KUKA KRL program: f1_Kuka_APT222T03S22.SRC

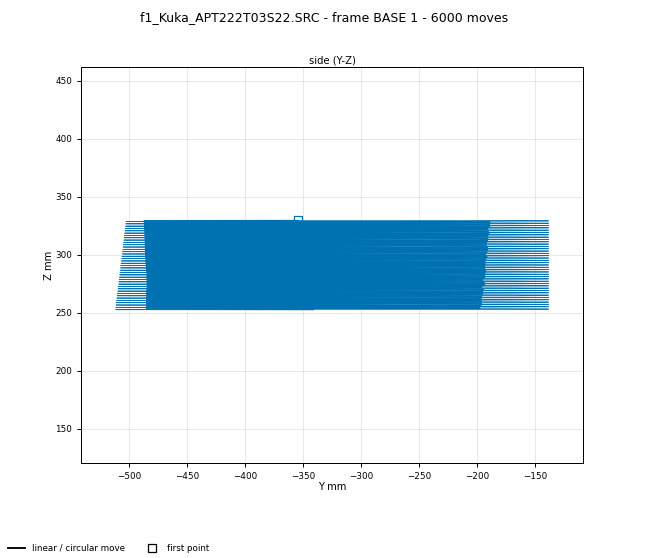
[picture p0: tool path of f1_Kuka_APT222T03S22.SRC in frame BASE 1, 6000 of 6001 moves have a stored position in this frame; points joined in program order, loops and branches not executed]
&ACCESS RVP
&REL 2
&PARAM TEMPLATE = C:\KRC\Roboter\Template\vorgabe
&PARAM EDITMASK = *
DEF f1_Kuka_APT222T03S22()


;FOLD INI;%{PE}%V3.2.0,%MKUKATPBASIS,%CINIT,%VCOMMON,%P
  ;FOLD BAS INI;%{E}%V3.2.0,%MKUKATPBASIS,%CINIT,%VINIT,%P
    GLOBAL INTERRUPT DECL 3 WHEN $STOPMESS==TRUE DO IR_STOPM ( )
    INTERRUPT ON 3
    BAS (#INITMOV,0 )
  ;ENDFOLD (BAS INI)
  ;FOLD USER INI;%{E}%V3.2.0,%MKUKATPUSER,%CINIT,%VINIT,%P
    ;Make your modifications here
  ;ENDFOLD (USER INI)
;ENDFOLD (INI)


;*** Make Null PTP Move
  PTP $pos_act

;*** Auto Load The Correct TOOL Data
  $tool=tool_data[3]

;*** Auto Load The Correct BASE Data
  $base=base_data[1]

  $ADVANCE = 5

;*** Restate Last Velocity
MMPM(30000.0)
SetRPM(6000)
LIN {X -0.045,Y -354.081,Z 329.624,A 0.000,B 0.000,C 90.000,E1 292.333} C_DIS
LIN {X -0.124,Y -370.125,Z 329.612,A 0.000,B 0.000,C 90.000,E1 290.248} C_DIS
LIN {X -0.194,Y -391.997,Z 329.598,A 0.000,B 0.000,C 90.000,E1 287.638} C_DIS
LIN {X 0.138,Y -406.942,Z 329.588,A 0.000,B 0.000,C 90.000,E1 285.898} C_DIS
LIN {X -0.099,Y -421.524,Z 329.579,A 0.000,B 0.000,C 90.000,E1 284.300} C_DIS
LIN {X 0.209,Y -431.131,Z 329.573,A 0.000,B 0.000,C 90.000,E1 283.175} C_DIS
LIN {X -0.088,Y -437.715,Z 329.569,A 0.000,B 0.000,C 90.000,E1 282.411} C_DIS
LIN {X -0.210,Y -445.768,Z 329.563,A 0.000,B 0.000,C 90.000,E1 281.366} C_DIS
LIN {X -0.147,Y -453.240,Z 329.557,A 0.000,B 0.000,C 90.000,E1 280.310} C_DIS
LIN {X -0.080,Y -460.078,Z 329.551,A 0.000,B 0.000,C 90.000,E1 279.265} C_DIS
LIN {X -0.164,Y -468.020,Z 329.544,A 0.000,B 0.000,C 90.000,E1 277.992} C_DIS
LIN {X 0.077,Y -473.919,Z 329.539,A 0.000,B 0.000,C 90.000,E1 276.947} C_DIS
LIN {X -0.147,Y -479.234,Z 329.533,A 0.000,B 0.000,C 90.000,E1 275.967} C_DIS
LIN {X -0.044,Y -481.494,Z 329.530,A 0.000,B 0.000,C 90.000,E1 275.454} C_DIS
LIN {X 0.122,Y -483.441,Z 329.527,A 0.000,B 0.000,C 90.000,E1 274.935} C_DIS
LIN {X -0.189,Y -484.967,Z 329.525,A 0.000,B 0.000,C 90.000,E1 274.473} C_DIS
LIN {X -0.009,Y -486.097,Z 329.522,A 0.000,B 0.000,C 90.000,E1 273.955} C_DIS
LIN {X 0.148,Y -486.777,Z 329.519,A 0.000,B 0.000,C 90.000,E1 273.440} C_DIS
LIN {X -0.146,Y -487.135,Z 329.516,A 0.000,B 0.000,C 90.000,E1 272.980} C_DIS
LIN {X 0.025,Y -487.164,Z 329.514,A 0.000,B 0.000,C 90.000,E1 272.465} C_DIS
LIN {X -0.093,Y -486.656,Z 329.508,A 0.000,B 0.000,C 90.000,E1 271.489} C_DIS
LIN {X 0.082,Y -486.195,Z 329.505,A 0.000,B 0.000,C 90.000,E1 270.974} C_DIS
LIN {X -0.228,Y -485.501,Z 329.503,A 0.000,B 0.000,C 90.000,E1 270.516} C_DIS
LIN {X -0.056,Y -484.497,Z 329.500,A 0.000,B 0.000,C 90.000,E1 270.000} C_DIS
LIN {X 0.112,Y -482.951,Z 329.497,A 0.000,B 0.000,C 90.000,E1 269.484} C_DIS
LIN {X -0.209,Y -480.802,Z 329.494,A 0.000,B 0.000,C 90.000,E1 269.026} C_DIS
LIN {X -0.057,Y -477.885,Z 329.492,A 0.000,B 0.000,C 90.000,E1 268.511} C_DIS
LIN {X -0.231,Y -476.129,Z 329.490,A 0.000,B 0.000,C 90.000,E1 268.282} C_DIS
LIN {X 0.087,Y -474.110,Z 329.489,A 0.000,B 0.000,C 90.000,E1 267.993} C_DIS
LIN {X 0.195,Y -469.213,Z 329.486,A 0.000,B 0.000,C 90.000,E1 267.478} C_DIS
LIN {X 0.065,Y -466.330,Z 329.485,A 0.000,B 0.000,C 90.000,E1 267.249} C_DIS
LIN {X -0.065,Y -463.081,Z 329.483,A 0.000,B 0.000,C 90.000,E1 267.020} C_DIS
LIN {X 0.146,Y -459.910,Z 329.482,A 0.000,B 0.000,C 90.000,E1 266.788} C_DIS
LIN {X -0.126,Y -456.229,Z 329.481,A 0.000,B 0.000,C 90.000,E1 266.617} C_DIS
LIN {X -0.058,Y -452.834,Z 329.480,A 0.000,B 0.000,C 90.000,E1 266.445} C_DIS
LIN {X -0.061,Y -445.345,Z 329.479,A 0.000,B 0.000,C 90.000,E1 266.159} C_DIS
LIN {X 0.071,Y -437.546,Z 329.477,A 0.000,B 0.000,C 90.000,E1 265.927} C_DIS
LIN {X 0.203,Y -429.002,Z 329.477,A 0.000,B 0.000,C 90.000,E1 265.755} C_DIS
LIN {X 0.032,Y -418.844,Z 329.476,A 0.000,B 0.000,C 90.000,E1 265.698} C_DIS
LIN {X -0.015,Y -180.910,Z 329.476,A 0.000,B 0.000,C 90.000,E1 265.698} C_DIS
LIN {X 0.075,Y -180.806,Z 329.471,A 0.000,B 0.000,C 90.000,E1 264.780} C_DIS
LIN {X -0.027,Y -178.907,Z 329.443,A 0.000,B 0.000,C 90.000,E1 259.746} C_DIS
LIN {X 0.053,Y -175.951,Z 329.415,A 0.000,B 0.000,C 90.000,E1 254.629} C_DIS
LIN {X 0.000,Y -175.416,Z 329.410,A 0.000,B 0.000,C 90.000,E1 253.795} C_DIS
LIN {X 0.003,Y -172.179,Z 329.386,A 0.000,B 0.000,C 90.000,E1 249.518} C_DIS
LIN {X 0.042,Y -171.650,Z 329.381,A 0.000,B 0.000,C 90.000,E1 248.646} C_DIS
LIN {X 0.036,Y -167.874,Z 329.357,A 0.000,B 0.000,C 90.000,E1 244.332} C_DIS
LIN {X -0.021,Y -166.608,Z 329.348,A 0.000,B 0.000,C 90.000,E1 242.615} C_DIS
LIN {X -0.027,Y -162.597,Z 329.324,A 0.000,B 0.000,C 90.000,E1 238.250} C_DIS
LIN {X -0.053,Y -161.281,Z 329.314,A 0.000,B 0.000,C 90.000,E1 236.501} C_DIS
LIN {X -0.017,Y -157.280,Z 329.289,A 0.000,B 0.000,C 90.000,E1 232.065} C_DIS
LIN {X 0.006,Y -155.999,Z 329.279,A 0.000,B 0.000,C 90.000,E1 230.275} C_DIS
LIN {X -0.034,Y -152.257,Z 329.254,A 0.000,B 0.000,C 90.000,E1 225.810} C_DIS
LIN {X -0.012,Y -150.495,Z 329.239,A 0.000,B 0.000,C 90.000,E1 223.095} C_DIS
LIN {X 0.018,Y -147.219,Z 329.214,A 0.000,B 0.000,C 90.000,E1 218.543} C_DIS
LIN {X -0.013,Y -145.241,Z 329.194,A 0.000,B 0.000,C 90.000,E1 214.898} C_DIS
LIN {X 0.029,Y -142.362,Z 329.163,A 0.000,B 0.000,C 90.000,E1 209.361} C_DIS
LIN {X 0.025,Y -141.748,Z 329.153,A 0.000,B 0.000,C 90.000,E1 207.513} C_DIS
LIN {X -0.048,Y -139.492,Z 329.117,A 0.000,B 0.000,C 90.000,E1 201.046} C_DIS
LIN {X -0.012,Y -138.995,Z 329.101,A 0.000,B 0.000,C 90.000,E1 198.236} C_DIS
LIN {X -0.055,Y -138.336,Z 329.055,A 0.000,B 0.000,C 90.000,E1 189.849} C_DIS
LIN {X -0.033,Y -139.415,Z 329.008,A 0.000,B 0.000,C 90.000,E1 181.432} C_DIS
LIN {X 0.021,Y -141.329,Z 328.972,A 0.000,B 0.000,C 90.000,E1 174.894} C_DIS
LIN {X -0.022,Y -142.686,Z 328.956,A 0.000,B 0.000,C 90.000,E1 172.129} C_DIS
LIN {X -0.043,Y -145.046,Z 328.931,A 0.000,B 0.000,C 90.000,E1 167.521} C_DIS
LIN {X -0.046,Y -147.673,Z 328.910,A 0.000,B 0.000,C 90.000,E1 163.850} C_DIS
LIN {X -0.011,Y -150.315,Z 328.890,A 0.000,B 0.000,C 90.000,E1 160.188} C_DIS
LIN {X 0.061,Y -153.728,Z 328.870,A 0.000,B 0.000,C 90.000,E1 156.538} C_DIS
LIN {X -0.087,Y -157.141,Z 328.850,A 0.000,B 0.000,C 90.000,E1 152.999} C_DIS
LIN {X -0.013,Y -161.290,Z 328.830,A 0.000,B 0.000,C 90.000,E1 149.410} C_DIS
LIN {X 0.004,Y -164.406,Z 328.815,A 0.000,B 0.000,C 90.000,E1 146.755} C_DIS
LIN {X 0.001,Y -169.087,Z 328.796,A 0.000,B 0.000,C 90.000,E1 143.256} C_DIS
LIN {X -0.048,Y -171.643,Z 328.786,A 0.000,B 0.000,C 90.000,E1 141.537} C_DIS
LIN {X -0.001,Y -176.606,Z 328.767,A 0.000,B 0.000,C 90.000,E1 138.081} C_DIS
LIN {X 0.000,Y -180.905,Z 328.753,A 0.000,B 0.000,C 90.000,E1 135.526} C_DIS
LIN {X -0.009,Y -186.320,Z 328.734,A 0.000,B 0.000,C 90.000,E1 132.162} C_DIS
LIN {X 0.058,Y -190.954,Z 328.720,A 0.000,B 0.000,C 90.000,E1 129.644} C_DIS
LIN {X -0.022,Y -196.725,Z 328.702,A 0.000,B 0.000,C 90.000,E1 126.377} C_DIS
LIN {X -0.054,Y -201.183,Z 328.689,A 0.000,B 0.000,C 90.000,E1 124.119} C_DIS
LIN {X -0.051,Y -201.261,Z 328.689,A 0.000,B 0.000,C 90.000,E1 124.072} C_DIS
LIN {X 0.058,Y -302.172,Z 328.689,A 0.000,B 0.000,C 90.000,E1 124.040} C_DIS
LIN {X 0.097,Y -306.283,Z 328.689,A 0.000,B 0.000,C 90.000,E1 123.913} C_DIS
LIN {X -0.045,Y -309.181,Z 328.687,A 0.000,B 0.000,C 90.000,E1 123.754} C_DIS
LIN {X -0.078,Y -312.923,Z 328.685,A 0.000,B 0.000,C 90.000,E1 123.372} C_DIS
LIN {X 0.156,Y -316.425,Z 328.682,A 0.000,B 0.000,C 90.000,E1 122.752} C_DIS
LIN {X 0.006,Y -318.957,Z 328.679,A 0.000,B 0.000,C 90.000,E1 122.133} C_DIS
LIN {X -0.076,Y -329.793,Z 328.663,A 0.000,B 0.000,C 90.000,E1 119.283} C_DIS
LIN {X -0.172,Y -342.027,Z 328.647,A 0.000,B 0.000,C 90.000,E1 116.488} C_DIS
LIN {X -0.094,Y -354.161,Z 328.633,A 0.000,B 0.000,C 90.000,E1 114.027} C_DIS
LIN {X 0.155,Y -367.575,Z 328.620,A 0.000,B 0.000,C 90.000,E1 111.589} C_DIS
LIN {X -0.007,Y -382.364,Z 328.607,A 0.000,B 0.000,C 90.000,E1 109.268} C_DIS
LIN {X -0.052,Y -398.640,Z 328.594,A 0.000,B 0.000,C 90.000,E1 106.985} C_DIS
LIN {X -0.199,Y -416.523,Z 328.582,A 0.000,B 0.000,C 90.000,E1 104.773} C_DIS
LIN {X -0.055,Y -436.052,Z 328.570,A 0.000,B 0.000,C 90.000,E1 102.591} C_DIS
LIN {X -0.147,Y -456.379,Z 328.559,A 0.000,B 0.000,C 90.000,E1 100.602} C_DIS
LIN {X 0.183,Y -479.856,Z 328.547,A 0.000,B 0.000,C 90.000,E1 98.511} C_DIS
LIN {X -0.219,Y -495.644,Z 328.540,A 0.000,B 0.000,C 90.000,E1 97.296} C_DIS
LIN {X -0.016,Y -497.526,Z 328.539,A 0.000,B 0.000,C 90.000,E1 97.068} C_DIS
LIN {X -0.103,Y -499.247,Z 328.538,A 0.000,B 0.000,C 90.000,E1 96.834} C_DIS
LIN {X -0.251,Y -500.536,Z 328.537,A 0.000,B 0.000,C 90.000,E1 96.606} C_DIS
LIN {X 0.032,Y -502.123,Z 328.534,A 0.000,B 0.000,C 90.000,E1 96.087} C_DIS
LIN {X -0.178,Y -502.633,Z 328.531,A 0.000,B 0.000,C 90.000,E1 95.625} C_DIS
LIN {X 0.120,Y -502.144,Z 328.528,A 0.000,B 0.000,C 90.000,E1 95.106} C_DIS
LIN {X -0.081,Y -500.573,Z 328.526,A 0.000,B 0.000,C 90.000,E1 94.645} C_DIS
LIN {X -0.202,Y -499.293,Z 328.524,A 0.000,B 0.000,C 90.000,E1 94.416} C_DIS
LIN {X -0.045,Y -494.012,Z 328.520,A 0.000,B 0.000,C 90.000,E1 93.669} C_DIS
LIN {X -0.084,Y -486.242,Z 328.515,A 0.000,B 0.000,C 90.000,E1 92.694} C_DIS
LIN {X -0.157,Y -467.875,Z 328.502,A 0.000,B 0.000,C 90.000,E1 90.458} C_DIS
LIN {X 0.002,Y -448.883,Z 328.488,A 0.000,B 0.000,C 90.000,E1 87.879} C_DIS
LIN {X -0.168,Y -430.026,Z 328.472,A 0.000,B 0.000,C 90.000,E1 85.008} C_DIS
LIN {X -0.089,Y -414.527,Z 328.457,A 0.000,B 0.000,C 90.000,E1 82.299} C_DIS
LIN {X 0.114,Y -399.996,Z 328.442,A 0.000,B 0.000,C 90.000,E1 79.511} C_DIS
LIN {X -0.212,Y -389.916,Z 328.431,A 0.000,B 0.000,C 90.000,E1 77.589} C_DIS
LIN {X -0.081,Y -378.252,Z 328.418,A 0.000,B 0.000,C 90.000,E1 75.283} C_DIS
LIN {X -0.109,Y -368.106,Z 328.407,A 0.000,B 0.000,C 90.000,E1 73.251} C_DIS
LIN {X 0.100,Y -357.919,Z 328.395,A 0.000,B 0.000,C 90.000,E1 71.148} C_DIS
LIN {X -0.103,Y -346.247,Z 328.382,A 0.000,B 0.000,C 90.000,E1 68.773} C_DIS
LIN {X 0.108,Y -333.824,Z 328.367,A 0.000,B 0.000,C 90.000,E1 65.973} C_DIS
LIN {X -0.011,Y -320.451,Z 328.347,A 0.000,B 0.000,C 90.000,E1 62.538} C_DIS
LIN {X -0.030,Y -309.036,Z 328.330,A 0.000,B 0.000,C 90.000,E1 59.331} C_DIS
LIN {X 0.011,Y -297.294,Z 328.310,A 0.000,B 0.000,C 90.000,E1 55.722} C_DIS
LIN {X -0.049,Y -287.389,Z 328.291,A 0.000,B 0.000,C 90.000,E1 52.396} C_DIS
LIN {X 0.036,Y -279.768,Z 328.276,A 0.000,B 0.000,C 90.000,E1 49.666} C_DIS
LIN {X -0.101,Y -274.008,Z 328.265,A 0.000,B 0.000,C 90.000,E1 47.634} C_DIS
LIN {X -0.035,Y -266.352,Z 328.249,A 0.000,B 0.000,C 90.000,E1 44.838} C_DIS
LIN {X 0.122,Y -260.736,Z 328.237,A 0.000,B 0.000,C 90.000,E1 42.690} C_DIS
LIN {X -0.176,Y -255.046,Z 328.225,A 0.000,B 0.000,C 90.000,E1 40.620} C_DIS
LIN {X 0.006,Y -249.323,Z 328.213,A 0.000,B 0.000,C 90.000,E1 38.418} C_DIS
LIN {X 0.075,Y -243.454,Z 328.201,A 0.000,B 0.000,C 90.000,E1 36.217} C_DIS
LIN {X -0.050,Y -235.570,Z 328.185,A 0.000,B 0.000,C 90.000,E1 33.293} C_DIS
LIN {X 0.092,Y -227.992,Z 328.168,A 0.000,B 0.000,C 90.000,E1 30.256} C_DIS
LIN {X -0.098,Y -220.827,Z 328.151,A 0.000,B 0.000,C 90.000,E1 27.257} C_DIS
LIN {X 0.024,Y -214.294,Z 328.134,A 0.000,B 0.000,C 90.000,E1 24.131} C_DIS
LIN {X 0.107,Y -208.616,Z 328.117,A 0.000,B 0.000,C 90.000,E1 20.972} C_DIS
LIN {X -0.040,Y -202.573,Z 328.095,A 0.000,B 0.000,C 90.000,E1 17.040} C_DIS
LIN {X -0.053,Y -198.494,Z 328.077,A 0.000,B 0.000,C 90.000,E1 13.828} C_DIS
LIN {X 0.096,Y -194.493,Z 328.054,A 0.000,B 0.000,C 90.000,E1 9.726} C_DIS
LIN {X 0.063,Y -191.104,Z 328.027,A 0.000,B 0.000,C 90.000,E1 4.821} C_DIS
LIN {X -0.006,Y -188.880,Z 327.988,A 0.000,B 0.000,C 90.000,E1 357.879} C_DIS
LIN {X 0.038,Y -190.678,Z 327.933,A 0.000,B 0.000,C 90.000,E1 347.937} C_DIS
LIN {X -0.017,Y -193.867,Z 327.906,A 0.000,B 0.000,C 90.000,E1 343.015} C_DIS
LIN {X 0.080,Y -197.691,Z 327.883,A 0.000,B 0.000,C 90.000,E1 338.901} C_DIS
LIN {X 0.105,Y -202.533,Z 327.860,A 0.000,B 0.000,C 90.000,E1 334.845} C_DIS
LIN {X -0.015,Y -208.379,Z 327.838,A 0.000,B 0.000,C 90.000,E1 330.873} C_DIS
LIN {X 0.008,Y -215.221,Z 327.816,A 0.000,B 0.000,C 90.000,E1 326.914} C_DIS
LIN {X 0.068,Y -222.764,Z 327.795,A 0.000,B 0.000,C 90.000,E1 323.004} C_DIS
LIN {X -0.004,Y -229.499,Z 327.777,A 0.000,B 0.000,C 90.000,E1 319.952} C_DIS
LIN {X 0.045,Y -238.222,Z 327.759,A 0.000,B 0.000,C 90.000,E1 316.539} C_DIS
LIN {X 0.014,Y -247.221,Z 327.742,A 0.000,B 0.000,C 90.000,E1 313.581} C_DIS
LIN {X 0.069,Y -258.416,Z 327.724,A 0.000,B 0.000,C 90.000,E1 310.297} C_DIS
LIN {X 0.015,Y -270.485,Z 327.706,A 0.000,B 0.000,C 90.000,E1 307.111} C_DIS
LIN {X -0.011,Y -279.232,Z 327.695,A 0.000,B 0.000,C 90.000,E1 305.025} C_DIS
LIN {X 0.126,Y -293.754,Z 327.678,A 0.000,B 0.000,C 90.000,E1 301.926} C_DIS
LIN {X 0.079,Y -309.866,Z 327.661,A 0.000,B 0.000,C 90.000,E1 298.949} C_DIS
LIN {X 0.106,Y -321.655,Z 327.650,A 0.000,B 0.000,C 90.000,E1 297.001} C_DIS
LIN {X -0.144,Y -338.816,Z 327.636,A 0.000,B 0.000,C 90.000,E1 294.515} C_DIS
LIN {X 0.065,Y -356.624,Z 327.622,A 0.000,B 0.000,C 90.000,E1 292.025} C_DIS
LIN {X 0.136,Y -375.134,Z 327.609,A 0.000,B 0.000,C 90.000,E1 289.631} C_DIS
LIN {X -0.123,Y -396.978,Z 327.595,A 0.000,B 0.000,C 90.000,E1 287.094} C_DIS
LIN {X -0.204,Y -411.779,Z 327.586,A 0.000,B 0.000,C 90.000,E1 285.426} C_DIS
LIN {X -0.152,Y -426.487,Z 327.576,A 0.000,B 0.000,C 90.000,E1 283.772} C_DIS
LIN {X 0.085,Y -433.401,Z 327.572,A 0.000,B 0.000,C 90.000,E1 282.939} C_DIS
LIN {X 0.004,Y -441.777,Z 327.566,A 0.000,B 0.000,C 90.000,E1 281.883} C_DIS
LIN {X -0.067,Y -449.482,Z 327.560,A 0.000,B 0.000,C 90.000,E1 280.838} C_DIS
LIN {X -0.040,Y -456.608,Z 327.554,A 0.000,B 0.000,C 90.000,E1 279.792} C_DIS
LIN {X -0.101,Y -464.753,Z 327.547,A 0.000,B 0.000,C 90.000,E1 278.511} C_DIS
LIN {X 0.041,Y -470.830,Z 327.542,A 0.000,B 0.000,C 90.000,E1 277.473} C_DIS
LIN {X -0.156,Y -476.468,Z 327.536,A 0.000,B 0.000,C 90.000,E1 276.486} C_DIS
LIN {X -0.213,Y -480.238,Z 327.532,A 0.000,B 0.000,C 90.000,E1 275.739} C_DIS
LIN {X -0.237,Y -483.273,Z 327.528,A 0.000,B 0.000,C 90.000,E1 274.992} C_DIS
LIN {X -0.068,Y -484.803,Z 327.525,A 0.000,B 0.000,C 90.000,E1 274.473} C_DIS
LIN {X 0.111,Y -485.920,Z 327.522,A 0.000,B 0.000,C 90.000,E1 273.955} C_DIS
LIN {X -0.219,Y -486.610,Z 327.519,A 0.000,B 0.000,C 90.000,E1 273.498} C_DIS
LIN {X -0.028,Y -486.989,Z 327.517,A 0.000,B 0.000,C 90.000,E1 272.980} C_DIS
LIN {X 0.142,Y -487.029,Z 327.514,A 0.000,B 0.000,C 90.000,E1 272.465} C_DIS
LIN {X 0.023,Y -486.519,Z 327.508,A 0.000,B 0.000,C 90.000,E1 271.489} C_DIS
LIN {X 0.197,Y -486.074,Z 327.506,A 0.000,B 0.000,C 90.000,E1 270.974} C_DIS
LIN {X -0.114,Y -485.390,Z 327.503,A 0.000,B 0.000,C 90.000,E1 270.516} C_DIS
LIN {X 0.057,Y -484.402,Z 327.500,A 0.000,B 0.000,C 90.000,E1 270.000} C_DIS
LIN {X 0.224,Y -482.871,Z 327.497,A 0.000,B 0.000,C 90.000,E1 269.484} C_DIS
LIN {X -0.097,Y -480.780,Z 327.495,A 0.000,B 0.000,C 90.000,E1 269.026} C_DIS
LIN {X 0.053,Y -477.912,Z 327.492,A 0.000,B 0.000,C 90.000,E1 268.511} C_DIS
LIN {X 0.196,Y -474.183,Z 327.489,A 0.000,B 0.000,C 90.000,E1 267.993} C_DIS
LIN {X -0.166,Y -469.376,Z 327.486,A 0.000,B 0.000,C 90.000,E1 267.535} C_DIS
LIN {X 0.163,Y -466.544,Z 327.485,A 0.000,B 0.000,C 90.000,E1 267.249} C_DIS
LIN {X 0.025,Y -463.317,Z 327.483,A 0.000,B 0.000,C 90.000,E1 267.020} C_DIS
LIN {X 0.223,Y -460.234,Z 327.482,A 0.000,B 0.000,C 90.000,E1 266.788} C_DIS
LIN {X -0.064,Y -456.610,Z 327.481,A 0.000,B 0.000,C 90.000,E1 266.617} C_DIS
LIN {X -0.022,Y -453.219,Z 327.480,A 0.000,B 0.000,C 90.000,E1 266.445} C_DIS
LIN {X -0.073,Y -445.673,Z 327.479,A 0.000,B 0.000,C 90.000,E1 266.159} C_DIS
LIN {X 0.032,Y -437.850,Z 327.477,A 0.000,B 0.000,C 90.000,E1 265.927} C_DIS
LIN {X 0.145,Y -429.297,Z 327.477,A 0.000,B 0.000,C 90.000,E1 265.755} C_DIS
LIN {X -0.046,Y -419.572,Z 327.476,A 0.000,B 0.000,C 90.000,E1 265.698} C_DIS
LIN {X -0.114,Y -416.030,Z 327.476,A 0.000,B 0.000,C 90.000,E1 265.698} C_DIS
LIN {X -0.081,Y -180.910,Z 327.476,A 0.000,B 0.000,C 90.000,E1 265.698} C_DIS
LIN {X 0.037,Y -180.802,Z 327.471,A 0.000,B 0.000,C 90.000,E1 264.780} C_DIS
LIN {X -0.066,Y -178.902,Z 327.443,A 0.000,B 0.000,C 90.000,E1 259.746} C_DIS
LIN {X 0.015,Y -175.945,Z 327.415,A 0.000,B 0.000,C 90.000,E1 254.629} C_DIS
LIN {X -0.039,Y -175.405,Z 327.410,A 0.000,B 0.000,C 90.000,E1 253.795} C_DIS
LIN {X -0.036,Y -172.171,Z 327.386,A 0.000,B 0.000,C 90.000,E1 249.518} C_DIS
LIN {X 0.004,Y -171.641,Z 327.381,A 0.000,B 0.000,C 90.000,E1 248.646} C_DIS
LIN {X -0.001,Y -167.864,Z 327.357,A 0.000,B 0.000,C 90.000,E1 244.332} C_DIS
LIN {X -0.058,Y -166.597,Z 327.348,A 0.000,B 0.000,C 90.000,E1 242.615} C_DIS
LIN {X 0.075,Y -162.587,Z 327.323,A 0.000,B 0.000,C 90.000,E1 238.201} C_DIS
LIN {X -0.089,Y -161.271,Z 327.314,A 0.000,B 0.000,C 90.000,E1 236.501} C_DIS
LIN {X 0.043,Y -157.270,Z 327.289,A 0.000,B 0.000,C 90.000,E1 232.029} C_DIS
LIN {X -0.030,Y -155.990,Z 327.279,A 0.000,B 0.000,C 90.000,E1 230.275} C_DIS
LIN {X -0.069,Y -152.247,Z 327.254,A 0.000,B 0.000,C 90.000,E1 225.810} C_DIS
LIN {X -0.047,Y -150.487,Z 327.239,A 0.000,B 0.000,C 90.000,E1 223.095} C_DIS
LIN {X -0.016,Y -147.211,Z 327.214,A 0.000,B 0.000,C 90.000,E1 218.543} C_DIS
LIN {X -0.047,Y -145.232,Z 327.194,A 0.000,B 0.000,C 90.000,E1 214.898} C_DIS
LIN {X 0.065,Y -142.356,Z 327.163,A 0.000,B 0.000,C 90.000,E1 209.333} C_DIS
LIN {X -0.008,Y -141.743,Z 327.153,A 0.000,B 0.000,C 90.000,E1 207.513} C_DIS
LIN {X -0.032,Y -139.489,Z 327.117,A 0.000,B 0.000,C 90.000,E1 201.025} C_DIS
LIN {X -0.044,Y -138.992,Z 327.101,A 0.000,B 0.000,C 90.000,E1 198.236} C_DIS
LIN {X 0.048,Y -138.336,Z 327.055,A 0.000,B 0.000,C 90.000,E1 189.792} C_DIS
LIN {X -0.066,Y -139.418,Z 327.008,A 0.000,B 0.000,C 90.000,E1 181.432} C_DIS
LIN {X -0.013,Y -141.335,Z 326.972,A 0.000,B 0.000,C 90.000,E1 174.894} C_DIS
LIN {X -0.056,Y -142.691,Z 326.956,A 0.000,B 0.000,C 90.000,E1 172.129} C_DIS
LIN {X 0.065,Y -145.055,Z 326.931,A 0.000,B 0.000,C 90.000,E1 167.465} C_DIS
LIN {X 0.062,Y -147.680,Z 326.910,A 0.000,B 0.000,C 90.000,E1 163.795} C_DIS
LIN {X -0.046,Y -150.326,Z 326.890,A 0.000,B 0.000,C 90.000,E1 160.188} C_DIS
LIN {X 0.025,Y -153.742,Z 326.870,A 0.000,B 0.000,C 90.000,E1 156.538} C_DIS
LIN {X 0.017,Y -157.155,Z 326.850,A 0.000,B 0.000,C 90.000,E1 152.948} C_DIS
LIN {X -0.049,Y -161.307,Z 326.830,A 0.000,B 0.000,C 90.000,E1 149.410} C_DIS
LIN {X -0.032,Y -164.422,Z 326.815,A 0.000,B 0.000,C 90.000,E1 146.755} C_DIS
LIN {X -0.036,Y -169.106,Z 326.796,A 0.000,B 0.000,C 90.000,E1 143.256} C_DIS
LIN {X -0.085,Y -171.661,Z 326.786,A 0.000,B 0.000,C 90.000,E1 141.537} C_DIS
LIN {X -0.040,Y -176.626,Z 326.767,A 0.000,B 0.000,C 90.000,E1 138.081} C_DIS
LIN {X 0.088,Y -180.923,Z 326.753,A 0.000,B 0.000,C 90.000,E1 135.486} C_DIS
LIN {X -0.049,Y -186.342,Z 326.734,A 0.000,B 0.000,C 90.000,E1 132.162} C_DIS
LIN {X 0.018,Y -190.974,Z 326.720,A 0.000,B 0.000,C 90.000,E1 129.644} C_DIS
LIN {X -0.063,Y -196.749,Z 326.702,A 0.000,B 0.000,C 90.000,E1 126.377} C_DIS
LIN {X -0.012,Y -201.162,Z 326.690,A 0.000,B 0.000,C 90.000,E1 124.119} C_DIS
LIN {X 0.012,Y -201.366,Z 326.689,A 0.000,B 0.000,C 90.000,E1 123.992} C_DIS
LIN {X -0.018,Y -302.297,Z 326.689,A 0.000,B 0.000,C 90.000,E1 123.992} C_DIS
LIN {X 0.034,Y -305.307,Z 326.688,A 0.000,B 0.000,C 90.000,E1 123.913} C_DIS
LIN {X -0.183,Y -308.457,Z 326.688,A 0.000,B 0.000,C 90.000,E1 123.785} C_DIS
LIN {X 0.025,Y -312.067,Z 326.686,A 0.000,B 0.000,C 90.000,E1 123.420} C_DIS
LIN {X 0.137,Y -315.668,Z 326.683,A 0.000,B 0.000,C 90.000,E1 122.880} C_DIS
LIN {X 0.193,Y -317.253,Z 326.681,A 0.000,B 0.000,C 90.000,E1 122.546} C_DIS
LIN {X -0.013,Y -330.566,Z 326.662,A 0.000,B 0.000,C 90.000,E1 119.077} C_DIS
LIN {X -0.087,Y -342.897,Z 326.646,A 0.000,B 0.000,C 90.000,E1 116.283} C_DIS
LIN {X 0.009,Y -355.126,Z 326.632,A 0.000,B 0.000,C 90.000,E1 113.823} C_DIS
LIN {X 0.143,Y -368.642,Z 326.619,A 0.000,B 0.000,C 90.000,E1 111.408} C_DIS
LIN {X 0.008,Y -383.542,Z 326.606,A 0.000,B 0.000,C 90.000,E1 109.087} C_DIS
LIN {X -0.005,Y -399.937,Z 326.593,A 0.000,B 0.000,C 90.000,E1 106.804} C_DIS
LIN {X -0.121,Y -417.949,Z 326.581,A 0.000,B 0.000,C 90.000,E1 104.592} C_DIS
LIN {X 0.097,Y -437.567,Z 326.569,A 0.000,B 0.000,C 90.000,E1 102.411} C_DIS
LIN {X 0.028,Y -457.937,Z 326.558,A 0.000,B 0.000,C 90.000,E1 100.433} C_DIS
LIN {X -0.006,Y -481.486,Z 326.547,A 0.000,B 0.000,C 90.000,E1 98.398} C_DIS
LIN {X -0.044,Y -494.774,Z 326.541,A 0.000,B 0.000,C 90.000,E1 97.352} C_DIS
LIN {X 0.152,Y -496.923,Z 326.540,A 0.000,B 0.000,C 90.000,E1 97.125} C_DIS
LIN {X 0.147,Y -498.786,Z 326.538,A 0.000,B 0.000,C 90.000,E1 96.891} C_DIS
LIN {X 0.081,Y -500.200,Z 326.537,A 0.000,B 0.000,C 90.000,E1 96.663} C_DIS
LIN {X -0.137,Y -502.077,Z 326.534,A 0.000,B 0.000,C 90.000,E1 96.201} C_DIS
LIN {X 0.151,Y -502.826,Z 326.532,A 0.000,B 0.000,C 90.000,E1 95.682} C_DIS
LIN {X -0.052,Y -502.569,Z 326.529,A 0.000,B 0.000,C 90.000,E1 95.220} C_DIS
LIN {X 0.246,Y -501.265,Z 326.526,A 0.000,B 0.000,C 90.000,E1 94.702} C_DIS
LIN {X 0.125,Y -500.154,Z 326.525,A 0.000,B 0.000,C 90.000,E1 94.473} C_DIS
LIN {X 0.005,Y -498.656,Z 326.524,A 0.000,B 0.000,C 90.000,E1 94.245} C_DIS
LIN {X 0.020,Y -491.314,Z 326.518,A 0.000,B 0.000,C 90.000,E1 93.269} C_DIS
LIN {X -0.047,Y -483.293,Z 326.513,A 0.000,B 0.000,C 90.000,E1 92.293} C_DIS
LIN {X -0.132,Y -461.131,Z 326.497,A 0.000,B 0.000,C 90.000,E1 89.542} C_DIS
LIN {X 0.088,Y -444.508,Z 326.484,A 0.000,B 0.000,C 90.000,E1 87.192} C_DIS
LIN {X -0.073,Y -424.476,Z 326.467,A 0.000,B 0.000,C 90.000,E1 84.033} C_DIS
LIN {X 0.000,Y -407.970,Z 326.450,A 0.000,B 0.000,C 90.000,E1 81.027} C_DIS
LIN {X -0.078,Y -396.513,Z 326.438,A 0.000,B 0.000,C 90.000,E1 78.814} C_DIS
LIN {X -0.009,Y -386.378,Z 326.427,A 0.000,B 0.000,C 90.000,E1 76.825} C_DIS
LIN {X 0.132,Y -373.298,Z 326.412,A 0.000,B 0.000,C 90.000,E1 74.212} C_DIS
LIN {X -0.007,Y -363.115,Z 326.401,A 0.000,B 0.000,C 90.000,E1 72.181} C_DIS
LIN {X -0.134,Y -352.912,Z 326.389,A 0.000,B 0.000,C 90.000,E1 70.115} C_DIS
LIN {X 0.011,Y -337.258,Z 326.371,A 0.000,B 0.000,C 90.000,E1 66.741} C_DIS
LIN {X -0.163,Y -327.096,Z 326.357,A 0.000,B 0.000,C 90.000,E1 64.280} C_DIS
LIN {X 0.072,Y -316.518,Z 326.341,A 0.000,B 0.000,C 90.000,E1 61.385} C_DIS
LIN {X 0.033,Y -306.428,Z 326.325,A 0.000,B 0.000,C 90.000,E1 58.486} C_DIS
LIN {X 0.136,Y -295.931,Z 326.307,A 0.000,B 0.000,C 90.000,E1 55.182} C_DIS
LIN {X 0.018,Y -286.111,Z 326.288,A 0.000,B 0.000,C 90.000,E1 51.859} C_DIS
LIN {X -0.007,Y -280.388,Z 326.277,A 0.000,B 0.000,C 90.000,E1 49.828} C_DIS
LIN {X 0.053,Y -274.623,Z 326.265,A 0.000,B 0.000,C 90.000,E1 47.757} C_DIS
LIN {X 0.079,Y -265.078,Z 326.246,A 0.000,B 0.000,C 90.000,E1 44.271} C_DIS
LIN {X 0.033,Y -259.460,Z 326.234,A 0.000,B 0.000,C 90.000,E1 42.162} C_DIS
LIN {X 0.133,Y -251.839,Z 326.218,A 0.000,B 0.000,C 90.000,E1 39.277} C_DIS
LIN {X -0.099,Y -246.077,Z 326.206,A 0.000,B 0.000,C 90.000,E1 37.156} C_DIS
LIN {X -0.046,Y -240.111,Z 326.194,A 0.000,B 0.000,C 90.000,E1 34.945} C_DIS
LIN {X 0.015,Y -232.347,Z 326.178,A 0.000,B 0.000,C 90.000,E1 31.957} C_DIS
LIN {X -0.014,Y -223.115,Z 326.157,A 0.000,B 0.000,C 90.000,E1 28.180} C_DIS
LIN {X 0.069,Y -216.364,Z 326.139,A 0.000,B 0.000,C 90.000,E1 25.079} C_DIS
LIN {X 0.012,Y -210.388,Z 326.122,A 0.000,B 0.000,C 90.000,E1 21.972} C_DIS
LIN {X 0.060,Y -204.099,Z 326.100,A 0.000,B 0.000,C 90.000,E1 18.000} C_DIS
LIN {X -0.009,Y -198.883,Z 326.078,A 0.000,B 0.000,C 90.000,E1 14.008} C_DIS
LIN {X -0.037,Y -194.813,Z 326.055,A 0.000,B 0.000,C 90.000,E1 9.962} C_DIS
LIN {X -0.033,Y -191.370,Z 326.028,A 0.000,B 0.000,C 90.000,E1 5.049} C_DIS
LIN {X -0.005,Y -189.021,Z 325.988,A 0.000,B 0.000,C 90.000,E1 357.879} C_DIS
LIN {X 0.050,Y -190.774,Z 325.933,A 0.000,B 0.000,C 90.000,E1 347.937} C_DIS
LIN {X -0.002,Y -193.956,Z 325.906,A 0.000,B 0.000,C 90.000,E1 343.015} C_DIS
LIN {X 0.098,Y -197.752,Z 325.883,A 0.000,B 0.000,C 90.000,E1 338.901} C_DIS
LIN {X 0.124,Y -202.573,Z 325.860,A 0.000,B 0.000,C 90.000,E1 334.845} C_DIS
LIN {X 0.006,Y -208.430,Z 325.838,A 0.000,B 0.000,C 90.000,E1 330.873} C_DIS
LIN {X 0.032,Y -215.231,Z 325.816,A 0.000,B 0.000,C 90.000,E1 326.914} C_DIS
LIN {X -0.086,Y -222.759,Z 325.795,A 0.000,B 0.000,C 90.000,E1 323.050} C_DIS
LIN {X -0.127,Y -229.497,Z 325.778,A 0.000,B 0.000,C 90.000,E1 319.989} C_DIS
LIN {X -0.057,Y -237.198,Z 325.761,A 0.000,B 0.000,C 90.000,E1 316.944} C_DIS
LIN {X 0.049,Y -246.075,Z 325.744,A 0.000,B 0.000,C 90.000,E1 313.947} C_DIS
LIN {X -0.096,Y -257.206,Z 325.726,A 0.000,B 0.000,C 90.000,E1 310.701} C_DIS
LIN {X 0.138,Y -269.195,Z 325.708,A 0.000,B 0.000,C 90.000,E1 307.443} C_DIS
LIN {X 0.026,Y -279.371,Z 325.695,A 0.000,B 0.000,C 90.000,E1 305.025} C_DIS
LIN {X 0.014,Y -293.919,Z 325.678,A 0.000,B 0.000,C 90.000,E1 301.957} C_DIS
LIN {X 0.092,Y -308.212,Z 325.663,A 0.000,B 0.000,C 90.000,E1 299.283} C_DIS
LIN {X 0.164,Y -321.927,Z 325.650,A 0.000,B 0.000,C 90.000,E1 297.001} C_DIS
LIN {X -0.077,Y -339.113,Z 325.636,A 0.000,B 0.000,C 90.000,E1 294.515} C_DIS
LIN {X 0.183,Y -359.216,Z 325.621,A 0.000,B 0.000,C 90.000,E1 291.716} C_DIS
LIN {X -0.039,Y -380.134,Z 325.606,A 0.000,B 0.000,C 90.000,E1 289.087} C_DIS
LIN {X -0.114,Y -399.786,Z 325.593,A 0.000,B 0.000,C 90.000,E1 286.804} C_DIS
LIN {X 0.120,Y -412.101,Z 325.585,A 0.000,B 0.000,C 90.000,E1 285.371} C_DIS
LIN {X -0.222,Y -426.745,Z 325.576,A 0.000,B 0.000,C 90.000,E1 283.772} C_DIS
LIN {X -0.040,Y -433.660,Z 325.572,A 0.000,B 0.000,C 90.000,E1 282.939} C_DIS
LIN {X -0.120,Y -441.944,Z 325.566,A 0.000,B 0.000,C 90.000,E1 281.883} C_DIS
LIN {X -0.191,Y -449.608,Z 325.560,A 0.000,B 0.000,C 90.000,E1 280.838} C_DIS
LIN {X -0.164,Y -456.688,Z 325.554,A 0.000,B 0.000,C 90.000,E1 279.792} C_DIS
LIN {X -0.226,Y -464.789,Z 325.547,A 0.000,B 0.000,C 90.000,E1 278.511} C_DIS
LIN {X 0.228,Y -472.242,Z 325.540,A 0.000,B 0.000,C 90.000,E1 277.182} C_DIS
LIN {X -0.008,Y -477.763,Z 325.534,A 0.000,B 0.000,C 90.000,E1 276.201} C_DIS
LIN {X -0.053,Y -481.252,Z 325.530,A 0.000,B 0.000,C 90.000,E1 275.454} C_DIS
LIN {X 0.113,Y -483.180,Z 325.527,A 0.000,B 0.000,C 90.000,E1 274.935} C_DIS
LIN {X -0.200,Y -484.726,Z 325.525,A 0.000,B 0.000,C 90.000,E1 274.473} C_DIS
LIN {X -0.022,Y -485.833,Z 325.522,A 0.000,B 0.000,C 90.000,E1 273.955} C_DIS
LIN {X 0.133,Y -486.525,Z 325.519,A 0.000,B 0.000,C 90.000,E1 273.440} C_DIS
LIN {X -0.162,Y -486.857,Z 325.516,A 0.000,B 0.000,C 90.000,E1 272.980} C_DIS
LIN {X 0.008,Y -486.888,Z 325.514,A 0.000,B 0.000,C 90.000,E1 272.465} C_DIS
LIN {X -0.113,Y -486.364,Z 325.508,A 0.000,B 0.000,C 90.000,E1 271.489} C_DIS
LIN {X 0.060,Y -485.887,Z 325.505,A 0.000,B 0.000,C 90.000,E1 270.974} C_DIS
LIN {X 0.233,Y -485.233,Z 325.503,A 0.000,B 0.000,C 90.000,E1 270.458} C_DIS
LIN {X -0.081,Y -484.222,Z 325.500,A 0.000,B 0.000,C 90.000,E1 270.000} C_DIS
LIN {X 0.085,Y -482.701,Z 325.497,A 0.000,B 0.000,C 90.000,E1 269.484} C_DIS
LIN {X -0.236,Y -480.606,Z 325.494,A 0.000,B 0.000,C 90.000,E1 269.026} C_DIS
LIN {X -0.086,Y -477.760,Z 325.492,A 0.000,B 0.000,C 90.000,E1 268.511} C_DIS
LIN {X 0.056,Y -473.994,Z 325.489,A 0.000,B 0.000,C 90.000,E1 267.993} C_DIS
LIN {X -0.125,Y -471.768,Z 325.487,A 0.000,B 0.000,C 90.000,E1 267.764} C_DIS
LIN {X 0.164,Y -469.223,Z 325.486,A 0.000,B 0.000,C 90.000,E1 267.478} C_DIS
LIN {X 0.030,Y -466.410,Z 325.485,A 0.000,B 0.000,C 90.000,E1 267.249} C_DIS
LIN {X -0.102,Y -463.237,Z 325.483,A 0.000,B 0.000,C 90.000,E1 267.020} C_DIS
LIN {X 0.079,Y -460.066,Z 325.482,A 0.000,B 0.000,C 90.000,E1 266.788} C_DIS
LIN {X -0.175,Y -453.061,Z 325.480,A 0.000,B 0.000,C 90.000,E1 266.445} C_DIS
LIN {X -0.213,Y -445.507,Z 325.479,A 0.000,B 0.000,C 90.000,E1 266.159} C_DIS
LIN {X -0.094,Y -437.743,Z 325.477,A 0.000,B 0.000,C 90.000,E1 265.927} C_DIS
LIN {X 0.032,Y -428.986,Z 325.476,A 0.000,B 0.000,C 90.000,E1 265.755} C_DIS
LIN {X -0.153,Y -419.076,Z 325.476,A 0.000,B 0.000,C 90.000,E1 265.698} C_DIS
LIN {X 0.084,Y -180.910,Z 325.476,A 0.000,B 0.000,C 90.000,E1 265.641} C_DIS
LIN {X -0.011,Y -180.796,Z 325.471,A 0.000,B 0.000,C 90.000,E1 264.780} C_DIS
LIN {X 0.063,Y -178.895,Z 325.443,A 0.000,B 0.000,C 90.000,E1 259.690} C_DIS
LIN {X -0.032,Y -175.939,Z 325.415,A 0.000,B 0.000,C 90.000,E1 254.629} C_DIS
LIN {X 0.083,Y -175.391,Z 325.410,A 0.000,B 0.000,C 90.000,E1 253.740} C_DIS
LIN {X -0.082,Y -172.162,Z 325.386,A 0.000,B 0.000,C 90.000,E1 249.518} C_DIS
LIN {X -0.043,Y -171.630,Z 325.381,A 0.000,B 0.000,C 90.000,E1 248.646} C_DIS
LIN {X -0.047,Y -167.852,Z 325.357,A 0.000,B 0.000,C 90.000,E1 244.332} C_DIS
LIN {X 0.044,Y -166.584,Z 325.348,A 0.000,B 0.000,C 90.000,E1 242.564} C_DIS
LIN {X 0.030,Y -162.574,Z 325.323,A 0.000,B 0.000,C 90.000,E1 238.201} C_DIS
LIN {X 0.090,Y -161.256,Z 325.314,A 0.000,B 0.000,C 90.000,E1 236.421} C_DIS
LIN {X 0.000,Y -157.258,Z 325.289,A 0.000,B 0.000,C 90.000,E1 232.029} C_DIS
LIN {X -0.074,Y -155.980,Z 325.279,A 0.000,B 0.000,C 90.000,E1 230.275} C_DIS
LIN {X -0.003,Y -152.235,Z 325.254,A 0.000,B 0.000,C 90.000,E1 225.769} C_DIS
LIN {X 0.013,Y -150.477,Z 325.239,A 0.000,B 0.000,C 90.000,E1 223.056} C_DIS
LIN {X -0.058,Y -147.202,Z 325.214,A 0.000,B 0.000,C 90.000,E1 218.543} C_DIS
LIN {X -0.005,Y -145.222,Z 325.194,A 0.000,B 0.000,C 90.000,E1 214.865} C_DIS
LIN {X 0.023,Y -142.350,Z 325.163,A 0.000,B 0.000,C 90.000,E1 209.333} C_DIS
LIN {X -0.050,Y -141.738,Z 325.153,A 0.000,B 0.000,C 90.000,E1 207.513} C_DIS
LIN {X 0.058,Y -139.486,Z 325.117,A 0.000,B 0.000,C 90.000,E1 200.972} C_DIS
LIN {X 0.047,Y -138.988,Z 325.101,A 0.000,B 0.000,C 90.000,E1 198.181} C_DIS
LIN {X 0.008,Y -138.335,Z 325.054,A 0.000,B 0.000,C 90.000,E1 189.792} C_DIS
LIN {X 0.032,Y -139.422,Z 325.008,A 0.000,B 0.000,C 90.000,E1 181.375} C_DIS
LIN {X -0.054,Y -141.343,Z 324.971,A 0.000,B 0.000,C 90.000,E1 174.894} C_DIS
LIN {X 0.063,Y -142.698,Z 324.956,A 0.000,B 0.000,C 90.000,E1 172.064} C_DIS
LIN {X 0.022,Y -145.065,Z 324.930,A 0.000,B 0.000,C 90.000,E1 167.465} C_DIS
LIN {X 0.019,Y -147.691,Z 324.910,A 0.000,B 0.000,C 90.000,E1 163.795} C_DIS
LIN {X -0.089,Y -150.340,Z 324.890,A 0.000,B 0.000,C 90.000,E1 160.188} C_DIS
LIN {X 0.046,Y -154.593,Z 324.865,A 0.000,B 0.000,C 90.000,E1 155.613} C_DIS
LIN {X 0.053,Y -158.132,Z 324.845,A 0.000,B 0.000,C 90.000,E1 152.025} C_DIS
LIN {X 0.014,Y -162.419,Z 324.825,A 0.000,B 0.000,C 90.000,E1 148.486} C_DIS
LIN {X -0.005,Y -166.675,Z 324.805,A 0.000,B 0.000,C 90.000,E1 144.975} C_DIS
LIN {X 0.001,Y -171.681,Z 324.786,A 0.000,B 0.000,C 90.000,E1 141.492} C_DIS
LIN {X -0.088,Y -176.650,Z 324.767,A 0.000,B 0.000,C 90.000,E1 138.081} C_DIS
LIN {X 0.040,Y -180.947,Z 324.753,A 0.000,B 0.000,C 90.000,E1 135.486} C_DIS
LIN {X 0.027,Y -186.368,Z 324.734,A 0.000,B 0.000,C 90.000,E1 132.123} C_DIS
LIN {X -0.032,Y -190.999,Z 324.720,A 0.000,B 0.000,C 90.000,E1 129.644} C_DIS
LIN {X -0.113,Y -196.776,Z 324.702,A 0.000,B 0.000,C 90.000,E1 126.377} C_DIS
LIN {X -0.077,Y -201.194,Z 324.689,A 0.000,B 0.000,C 90.000,E1 124.119} C_DIS
LIN {X 0.083,Y -201.468,Z 324.689,A 0.000,B 0.000,C 90.000,E1 123.913} C_DIS
LIN {X 0.082,Y -302.597,Z 324.688,A 0.000,B 0.000,C 90.000,E1 123.913} C_DIS
LIN {X -0.044,Y -304.031,Z 324.688,A 0.000,B 0.000,C 90.000,E1 123.913} C_DIS
LIN {X -0.083,Y -307.416,Z 324.688,A 0.000,B 0.000,C 90.000,E1 123.785} C_DIS
LIN {X 0.120,Y -310.752,Z 324.686,A 0.000,B 0.000,C 90.000,E1 123.499} C_DIS
LIN {X -0.038,Y -314.439,Z 324.684,A 0.000,B 0.000,C 90.000,E1 123.086} C_DIS
LIN {X 0.033,Y -316.320,Z 324.682,A 0.000,B 0.000,C 90.000,E1 122.752} C_DIS
LIN {X 0.105,Y -317.794,Z 324.680,A 0.000,B 0.000,C 90.000,E1 122.418} C_DIS
LIN {X -0.183,Y -329.825,Z 324.663,A 0.000,B 0.000,C 90.000,E1 119.283} C_DIS
LIN {X 0.028,Y -342.065,Z 324.647,A 0.000,B 0.000,C 90.000,E1 116.437} C_DIS
LIN {X -0.059,Y -354.208,Z 324.633,A 0.000,B 0.000,C 90.000,E1 114.003} C_DIS
LIN {X 0.044,Y -367.630,Z 324.620,A 0.000,B 0.000,C 90.000,E1 111.589} C_DIS
LIN {X -0.121,Y -382.430,Z 324.607,A 0.000,B 0.000,C 90.000,E1 109.268} C_DIS
LIN {X -0.053,Y -398.716,Z 324.594,A 0.000,B 0.000,C 90.000,E1 106.968} C_DIS
LIN {X 0.083,Y -416.611,Z 324.582,A 0.000,B 0.000,C 90.000,E1 104.717} C_DIS
LIN {X -0.165,Y -436.133,Z 324.570,A 0.000,B 0.000,C 90.000,E1 102.591} C_DIS
LIN {X 0.194,Y -456.465,Z 324.559,A 0.000,B 0.000,C 90.000,E1 100.546} C_DIS
LIN {X 0.058,Y -479.975,Z 324.547,A 0.000,B 0.000,C 90.000,E1 98.511} C_DIS
LIN {X 0.150,Y -495.821,Z 324.540,A 0.000,B 0.000,C 90.000,E1 97.239} C_DIS
LIN {X -0.010,Y -499.377,Z 324.538,A 0.000,B 0.000,C 90.000,E1 96.834} C_DIS
LIN {X -0.156,Y -500.744,Z 324.537,A 0.000,B 0.000,C 90.000,E1 96.606} C_DIS
LIN {X 0.253,Y -501.752,Z 324.535,A 0.000,B 0.000,C 90.000,E1 96.315} C_DIS
LIN {X 0.043,Y -502.884,Z 324.533,A 0.000,B 0.000,C 90.000,E1 95.853} C_DIS
LIN {X -0.163,Y -502.991,Z 324.530,A 0.000,B 0.000,C 90.000,E1 95.391} C_DIS
LIN {X 0.093,Y -502.086,Z 324.527,A 0.000,B 0.000,C 90.000,E1 94.878} C_DIS
LIN {X -0.105,Y -500.005,Z 324.524,A 0.000,B 0.000,C 90.000,E1 94.416} C_DIS
LIN {X 0.186,Y -496.625,Z 324.522,A 0.000,B 0.000,C 90.000,E1 93.898} C_DIS
LIN {X 0.172,Y -489.016,Z 324.516,A 0.000,B 0.000,C 90.000,E1 92.922} C_DIS
LIN {X -0.094,Y -478.784,Z 324.509,A 0.000,B 0.000,C 90.000,E1 91.718} C_DIS
LIN {X 0.137,Y -456.946,Z 324.494,A 0.000,B 0.000,C 90.000,E1 88.912} C_DIS
LIN {X -0.184,Y -440.706,Z 324.481,A 0.000,B 0.000,C 90.000,E1 86.617} C_DIS
LIN {X 0.162,Y -424.191,Z 324.466,A 0.000,B 0.000,C 90.000,E1 83.913} C_DIS
LIN {X -0.229,Y -407.714,Z 324.450,A 0.000,B 0.000,C 90.000,E1 80.971} C_DIS
LIN {X 0.080,Y -396.262,Z 324.437,A 0.000,B 0.000,C 90.000,E1 78.701} C_DIS
LIN {X -0.158,Y -386.114,Z 324.426,A 0.000,B 0.000,C 90.000,E1 76.756} C_DIS
LIN {X -0.104,Y -373.046,Z 324.412,A 0.000,B 0.000,C 90.000,E1 74.157} C_DIS
LIN {X 0.096,Y -362.887,Z 324.400,A 0.000,B 0.000,C 90.000,E1 72.072} C_DIS
LIN {X -0.042,Y -352.686,Z 324.389,A 0.000,B 0.000,C 90.000,E1 70.007} C_DIS
LIN {X -0.104,Y -337.059,Z 324.370,A 0.000,B 0.000,C 90.000,E1 66.666} C_DIS
LIN {X -0.015,Y -325.760,Z 324.355,A 0.000,B 0.000,C 90.000,E1 63.845} C_DIS
LIN {X -0.026,Y -316.406,Z 324.341,A 0.000,B 0.000,C 90.000,E1 61.307} C_DIS
LIN {X -0.107,Y -307.432,Z 324.326,A 0.000,B 0.000,C 90.000,E1 58.742} C_DIS
LIN {X -0.130,Y -296.867,Z 324.308,A 0.000,B 0.000,C 90.000,E1 55.468} C_DIS
LIN {X -0.035,Y -287.008,Z 324.289,A 0.000,B 0.000,C 90.000,E1 52.110} C_DIS
LIN {X 0.038,Y -279.342,Z 324.274,A 0.000,B 0.000,C 90.000,E1 49.380} C_DIS
LIN {X 0.075,Y -273.557,Z 324.263,A 0.000,B 0.000,C 90.000,E1 47.310} C_DIS
LIN {X -0.126,Y -264.060,Z 324.244,A 0.000,B 0.000,C 90.000,E1 43.866} C_DIS
LIN {X 0.004,Y -258.424,Z 324.232,A 0.000,B 0.000,C 90.000,E1 41.714} C_DIS
LIN {X 0.081,Y -250.803,Z 324.216,A 0.000,B 0.000,C 90.000,E1 38.830} C_DIS
LIN {X 0.026,Y -245.033,Z 324.204,A 0.000,B 0.000,C 90.000,E1 36.664} C_DIS
LIN {X 0.079,Y -237.089,Z 324.187,A 0.000,B 0.000,C 90.000,E1 33.706} C_DIS
LIN {X 0.059,Y -229.437,Z 324.171,A 0.000,B 0.000,C 90.000,E1 30.718} C_DIS
LIN {X -0.095,Y -222.146,Z 324.154,A 0.000,B 0.000,C 90.000,E1 27.719} C_DIS
LIN {X 0.066,Y -215.500,Z 324.137,A 0.000,B 0.000,C 90.000,E1 24.591} C_DIS
LIN {X 0.070,Y -209.667,Z 324.119,A 0.000,B 0.000,C 90.000,E1 21.461} C_DIS
LIN {X 0.018,Y -203.525,Z 324.097,A 0.000,B 0.000,C 90.000,E1 17.511} C_DIS
LIN {X 0.071,Y -198.479,Z 324.075,A 0.000,B 0.000,C 90.000,E1 13.480} C_DIS
LIN {X -0.005,Y -194.547,Z 324.052,A 0.000,B 0.000,C 90.000,E1 9.443} C_DIS
LIN {X -0.008,Y -191.251,Z 324.025,A 0.000,B 0.000,C 90.000,E1 4.531} C_DIS
LIN {X -0.087,Y -189.094,Z 323.984,A 0.000,B 0.000,C 90.000,E1 357.078} C_DIS
LIN {X 0.061,Y -190.885,Z 323.933,A 0.000,B 0.000,C 90.000,E1 347.937} C_DIS
LIN {X 0.014,Y -194.044,Z 323.906,A 0.000,B 0.000,C 90.000,E1 343.015} C_DIS
LIN {X -0.068,Y -197.830,Z 323.883,A 0.000,B 0.000,C 90.000,E1 338.954} C_DIS
LIN {X -0.038,Y -202.625,Z 323.860,A 0.000,B 0.000,C 90.000,E1 334.897} C_DIS
LIN {X 0.030,Y -208.474,Z 323.838,A 0.000,B 0.000,C 90.000,E1 330.873} C_DIS
LIN {X 0.057,Y -215.237,Z 323.816,A 0.000,B 0.000,C 90.000,E1 326.914} C_DIS
LIN {X -0.059,Y -222.756,Z 323.795,A 0.000,B 0.000,C 90.000,E1 323.050} C_DIS
LIN {X -0.100,Y -229.495,Z 323.778,A 0.000,B 0.000,C 90.000,E1 319.989} C_DIS
LIN {X -0.030,Y -237.234,Z 323.761,A 0.000,B 0.000,C 90.000,E1 316.944} C_DIS
LIN {X 0.079,Y -246.128,Z 323.744,A 0.000,B 0.000,C 90.000,E1 313.947} C_DIS
LIN {X -0.063,Y -257.276,Z 323.726,A 0.000,B 0.000,C 90.000,E1 310.701} C_DIS
LIN {X 0.175,Y -269.301,Z 323.708,A 0.000,B 0.000,C 90.000,E1 307.443} C_DIS
LIN {X 0.007,Y -281.057,Z 323.693,A 0.000,B 0.000,C 90.000,E1 304.692} C_DIS
LIN {X 0.061,Y -294.086,Z 323.678,A 0.000,B 0.000,C 90.000,E1 301.957} C_DIS
LIN {X -0.147,Y -306.581,Z 323.665,A 0.000,B 0.000,C 90.000,E1 299.667} C_DIS
LIN {X -0.132,Y -320.148,Z 323.652,A 0.000,B 0.000,C 90.000,E1 297.385} C_DIS
LIN {X -0.005,Y -339.398,Z 323.636,A 0.000,B 0.000,C 90.000,E1 294.515} C_DIS
LIN {X -0.066,Y -359.506,Z 323.621,A 0.000,B 0.000,C 90.000,E1 291.770} C_DIS
LIN {X 0.053,Y -380.363,Z 323.606,A 0.000,B 0.000,C 90.000,E1 289.087} C_DIS
LIN {X -0.018,Y -399.946,Z 323.593,A 0.000,B 0.000,C 90.000,E1 286.804} C_DIS
LIN {X -0.056,Y -414.635,Z 323.584,A 0.000,B 0.000,C 90.000,E1 285.134} C_DIS
LIN {X -0.106,Y -426.779,Z 323.576,A 0.000,B 0.000,C 90.000,E1 283.772} C_DIS
LIN {X 0.079,Y -433.629,Z 323.572,A 0.000,B 0.000,C 90.000,E1 282.939} C_DIS
LIN {X 0.001,Y -441.887,Z 323.566,A 0.000,B 0.000,C 90.000,E1 281.883} C_DIS
LIN {X -0.068,Y -449.529,Z 323.560,A 0.000,B 0.000,C 90.000,E1 280.838} C_DIS
LIN {X -0.041,Y -456.568,Z 323.554,A 0.000,B 0.000,C 90.000,E1 279.792} C_DIS
LIN {X 0.073,Y -463.077,Z 323.549,A 0.000,B 0.000,C 90.000,E1 278.746} C_DIS
LIN {X 0.039,Y -470.611,Z 323.542,A 0.000,B 0.000,C 90.000,E1 277.473} C_DIS
LIN {X -0.162,Y -476.267,Z 323.536,A 0.000,B 0.000,C 90.000,E1 276.486} C_DIS
LIN {X -0.221,Y -479.998,Z 323.532,A 0.000,B 0.000,C 90.000,E1 275.739} C_DIS
LIN {X -0.247,Y -482.994,Z 323.528,A 0.000,B 0.000,C 90.000,E1 274.992} C_DIS
LIN {X -0.079,Y -484.548,Z 323.525,A 0.000,B 0.000,C 90.000,E1 274.473} C_DIS
LIN {X 0.098,Y -485.680,Z 323.522,A 0.000,B 0.000,C 90.000,E1 273.955} C_DIS
LIN {X -0.233,Y -486.385,Z 323.519,A 0.000,B 0.000,C 90.000,E1 273.498} C_DIS
LIN {X -0.043,Y -486.702,Z 323.517,A 0.000,B 0.000,C 90.000,E1 272.980} C_DIS
LIN {X 0.126,Y -486.745,Z 323.514,A 0.000,B 0.000,C 90.000,E1 272.465} C_DIS
LIN {X 0.002,Y -486.246,Z 323.508,A 0.000,B 0.000,C 90.000,E1 271.489} C_DIS
LIN {X -0.138,Y -485.112,Z 323.503,A 0.000,B 0.000,C 90.000,E1 270.516} C_DIS
LIN {X 0.032,Y -484.111,Z 323.500,A 0.000,B 0.000,C 90.000,E1 270.000} C_DIS
LIN {X 0.197,Y -482.619,Z 323.497,A 0.000,B 0.000,C 90.000,E1 269.484} C_DIS
LIN {X -0.125,Y -480.546,Z 323.495,A 0.000,B 0.000,C 90.000,E1 269.026} C_DIS
LIN {X 0.023,Y -477.789,Z 323.492,A 0.000,B 0.000,C 90.000,E1 268.511} C_DIS
LIN {X 0.166,Y -474.126,Z 323.489,A 0.000,B 0.000,C 90.000,E1 267.993} C_DIS
LIN {X -0.196,Y -469.428,Z 323.486,A 0.000,B 0.000,C 90.000,E1 267.535} C_DIS
LIN {X -0.059,Y -463.408,Z 323.483,A 0.000,B 0.000,C 90.000,E1 267.020} C_DIS
LIN {X 0.091,Y -460.283,Z 323.482,A 0.000,B 0.000,C 90.000,E1 266.788} C_DIS
LIN {X 0.215,Y -456.624,Z 323.481,A 0.000,B 0.000,C 90.000,E1 266.560} C_DIS
LIN {X -0.219,Y -453.201,Z 323.480,A 0.000,B 0.000,C 90.000,E1 266.445} C_DIS
LIN {X 0.161,Y -445.565,Z 323.478,A 0.000,B 0.000,C 90.000,E1 266.102} C_DIS
LIN {X -0.189,Y -437.713,Z 323.477,A 0.000,B 0.000,C 90.000,E1 265.927} C_DIS
LIN {X -0.090,Y -428.600,Z 323.476,A 0.000,B 0.000,C 90.000,E1 265.755} C_DIS
LIN {X 0.143,Y -418.197,Z 323.476,A 0.000,B 0.000,C 90.000,E1 265.641} C_DIS
LIN {X 0.032,Y -180.909,Z 323.476,A 0.000,B 0.000,C 90.000,E1 265.641} C_DIS
LIN {X -0.061,Y -180.790,Z 323.471,A 0.000,B 0.000,C 90.000,E1 264.780} C_DIS
LIN {X 0.014,Y -178.889,Z 323.443,A 0.000,B 0.000,C 90.000,E1 259.690} C_DIS
LIN {X 0.089,Y -175.931,Z 323.414,A 0.000,B 0.000,C 90.000,E1 254.574} C_DIS
LIN {X 0.034,Y -175.378,Z 323.410,A 0.000,B 0.000,C 90.000,E1 253.740} C_DIS
LIN {X 0.032,Y -172.152,Z 323.386,A 0.000,B 0.000,C 90.000,E1 249.464} C_DIS
LIN {X 0.069,Y -171.617,Z 323.381,A 0.000,B 0.000,C 90.000,E1 248.592} C_DIS
LIN {X 0.057,Y -167.840,Z 323.357,A 0.000,B 0.000,C 90.000,E1 244.280} C_DIS
LIN {X -0.003,Y -166.569,Z 323.348,A 0.000,B 0.000,C 90.000,E1 242.564} C_DIS
LIN {X -0.016,Y -162.562,Z 323.323,A 0.000,B 0.000,C 90.000,E1 238.201} C_DIS
LIN {X 0.044,Y -161.242,Z 323.314,A 0.000,B 0.000,C 90.000,E1 236.421} C_DIS
LIN {X -0.045,Y -157.245,Z 323.289,A 0.000,B 0.000,C 90.000,E1 232.029} C_DIS
LIN {X 0.001,Y -155.969,Z 323.279,A 0.000,B 0.000,C 90.000,E1 230.231} C_DIS
LIN {X 0.059,Y -152.223,Z 323.254,A 0.000,B 0.000,C 90.000,E1 225.729} C_DIS
LIN {X -0.031,Y -150.466,Z 323.239,A 0.000,B 0.000,C 90.000,E1 223.056} C_DIS
LIN {X -0.011,Y -147.191,Z 323.214,A 0.000,B 0.000,C 90.000,E1 218.508} C_DIS
LIN {X 0.071,Y -145.210,Z 323.194,A 0.000,B 0.000,C 90.000,E1 214.818} C_DIS
LIN {X -0.020,Y -142.343,Z 323.163,A 0.000,B 0.000,C 90.000,E1 209.333} C_DIS
LIN {X 0.033,Y -141.731,Z 323.153,A 0.000,B 0.000,C 90.000,E1 207.462} C_DIS
LIN {X 0.015,Y -139.482,Z 323.117,A 0.000,B 0.000,C 90.000,E1 200.972} C_DIS
LIN {X 0.004,Y -138.982,Z 323.101,A 0.000,B 0.000,C 90.000,E1 198.181} C_DIS
LIN {X -0.034,Y -138.333,Z 323.054,A 0.000,B 0.000,C 90.000,E1 189.792} C_DIS
LIN {X -0.010,Y -139.426,Z 323.008,A 0.000,B 0.000,C 90.000,E1 181.375} C_DIS
LIN {X 0.044,Y -141.351,Z 322.971,A 0.000,B 0.000,C 90.000,E1 174.837} C_DIS
LIN {X 0.020,Y -142.705,Z 322.956,A 0.000,B 0.000,C 90.000,E1 172.064} C_DIS
LIN {X -0.021,Y -145.077,Z 322.930,A 0.000,B 0.000,C 90.000,E1 167.465} C_DIS
LIN {X -0.025,Y -147.701,Z 322.910,A 0.000,B 0.000,C 90.000,E1 163.795} C_DIS
LIN {X 0.008,Y -150.354,Z 322.890,A 0.000,B 0.000,C 90.000,E1 160.134} C_DIS
LIN {X 0.001,Y -154.608,Z 322.865,A 0.000,B 0.000,C 90.000,E1 155.613} C_DIS
LIN {X 0.008,Y -158.151,Z 322.845,A 0.000,B 0.000,C 90.000,E1 152.025} C_DIS
LIN {X 0.052,Y -162.436,Z 322.825,A 0.000,B 0.000,C 90.000,E1 148.456} C_DIS
LIN {X -0.052,Y -166.697,Z 322.805,A 0.000,B 0.000,C 90.000,E1 144.975} C_DIS
LIN {X 0.061,Y -171.702,Z 322.786,A 0.000,B 0.000,C 90.000,E1 141.457} C_DIS
LIN {X -0.005,Y -176.675,Z 322.767,A 0.000,B 0.000,C 90.000,E1 138.038} C_DIS
LIN {X -0.010,Y -180.972,Z 322.753,A 0.000,B 0.000,C 90.000,E1 135.486} C_DIS
LIN {X -0.024,Y -186.396,Z 322.734,A 0.000,B 0.000,C 90.000,E1 132.123} C_DIS
LIN {X -0.083,Y -191.024,Z 322.720,A 0.000,B 0.000,C 90.000,E1 129.644} C_DIS
LIN {X 0.109,Y -196.806,Z 322.702,A 0.000,B 0.000,C 90.000,E1 126.297} C_DIS
LIN {X 0.028,Y -200.059,Z 322.693,A 0.000,B 0.000,C 90.000,E1 124.692} C_DIS
LIN {X 0.038,Y -201.571,Z 322.688,A 0.000,B 0.000,C 90.000,E1 123.865} C_DIS
LIN {X 0.022,Y -302.910,Z 322.688,A 0.000,B 0.000,C 90.000,E1 123.865} C_DIS
LIN {X -0.063,Y -305.124,Z 322.688,A 0.000,B 0.000,C 90.000,E1 123.833} C_DIS
LIN {X 0.054,Y -308.818,Z 322.687,A 0.000,B 0.000,C 90.000,E1 123.627} C_DIS
LIN {X -0.001,Y -311.078,Z 322.686,A 0.000,B 0.000,C 90.000,E1 123.452} C_DIS
LIN {X -0.025,Y -314.223,Z 322.684,A 0.000,B 0.000,C 90.000,E1 123.086} C_DIS
LIN {X 0.070,Y -316.170,Z 322.682,A 0.000,B 0.000,C 90.000,E1 122.752} C_DIS
LIN {X -0.101,Y -317.692,Z 322.680,A 0.000,B 0.000,C 90.000,E1 122.467} C_DIS
LIN {X -0.011,Y -331.047,Z 322.661,A 0.000,B 0.000,C 90.000,E1 118.949} C_DIS
LIN {X -0.074,Y -343.446,Z 322.645,A 0.000,B 0.000,C 90.000,E1 116.155} C_DIS
LIN {X 0.035,Y -355.739,Z 322.632,A 0.000,B 0.000,C 90.000,E1 113.695} C_DIS
LIN {X 0.184,Y -369.322,Z 322.618,A 0.000,B 0.000,C 90.000,E1 111.280} C_DIS
LIN {X 0.064,Y -384.296,Z 322.605,A 0.000,B 0.000,C 90.000,E1 108.960} C_DIS
LIN {X 0.066,Y -400.770,Z 322.593,A 0.000,B 0.000,C 90.000,E1 106.677} C_DIS
LIN {X -0.138,Y -418.868,Z 322.580,A 0.000,B 0.000,C 90.000,E1 104.481} C_DIS
LIN {X 0.133,Y -438.550,Z 322.568,A 0.000,B 0.000,C 90.000,E1 102.299} C_DIS
LIN {X 0.226,Y -458.949,Z 322.557,A 0.000,B 0.000,C 90.000,E1 100.310} C_DIS
LIN {X -0.193,Y -482.497,Z 322.546,A 0.000,B 0.000,C 90.000,E1 98.333} C_DIS
LIN {X 0.203,Y -495.759,Z 322.540,A 0.000,B 0.000,C 90.000,E1 97.239} C_DIS
LIN {X 0.091,Y -499.395,Z 322.538,A 0.000,B 0.000,C 90.000,E1 96.834} C_DIS
LIN {X -0.056,Y -500.814,Z 322.537,A 0.000,B 0.000,C 90.000,E1 96.606} C_DIS
LIN {X -0.146,Y -501.865,Z 322.535,A 0.000,B 0.000,C 90.000,E1 96.372} C_DIS
LIN {X 0.144,Y -503.066,Z 322.533,A 0.000,B 0.000,C 90.000,E1 95.853} C_DIS
LIN {X -0.061,Y -503.236,Z 322.530,A 0.000,B 0.000,C 90.000,E1 95.391} C_DIS
LIN {X 0.196,Y -502.395,Z 322.527,A 0.000,B 0.000,C 90.000,E1 94.878} C_DIS
LIN {X -0.001,Y -500.397,Z 322.525,A 0.000,B 0.000,C 90.000,E1 94.416} C_DIS
LIN {X -0.205,Y -497.076,Z 322.522,A 0.000,B 0.000,C 90.000,E1 93.955} C_DIS
LIN {X -0.209,Y -489.455,Z 322.516,A 0.000,B 0.000,C 90.000,E1 92.980} C_DIS
LIN {X -0.146,Y -477.161,Z 322.508,A 0.000,B 0.000,C 90.000,E1 91.489} C_DIS
LIN {X 0.034,Y -455.443,Z 322.493,A 0.000,B 0.000,C 90.000,E1 88.682} C_DIS
LIN {X 0.122,Y -439.334,Z 322.480,A 0.000,B 0.000,C 90.000,E1 86.331} C_DIS
LIN {X -0.130,Y -424.525,Z 322.466,A 0.000,B 0.000,C 90.000,E1 83.970} C_DIS
LIN {X 0.017,Y -406.574,Z 322.448,A 0.000,B 0.000,C 90.000,E1 80.679} C_DIS
LIN {X -0.170,Y -396.579,Z 322.437,A 0.000,B 0.000,C 90.000,E1 78.757} C_DIS
LIN {X -0.016,Y -386.434,Z 322.426,A 0.000,B 0.000,C 90.000,E1 76.756} C_DIS
LIN {X 0.042,Y -373.383,Z 322.412,A 0.000,B 0.000,C 90.000,E1 74.157} C_DIS
LIN {X -0.101,Y -363.221,Z 322.401,A 0.000,B 0.000,C 90.000,E1 72.127} C_DIS
LIN {X 0.110,Y -353.032,Z 322.389,A 0.000,B 0.000,C 90.000,E1 70.007} C_DIS
LIN {X 0.052,Y -337.400,Z 322.370,A 0.000,B 0.000,C 90.000,E1 66.666} C_DIS
LIN {X -0.113,Y -327.295,Z 322.357,A 0.000,B 0.000,C 90.000,E1 64.204} C_DIS
LIN {X 0.057,Y -317.902,Z 322.342,A 0.000,B 0.000,C 90.000,E1 61.641} C_DIS
LIN {X 0.060,Y -307.784,Z 322.326,A 0.000,B 0.000,C 90.000,E1 58.742} C_DIS
LIN {X 0.043,Y -297.204,Z 322.308,A 0.000,B 0.000,C 90.000,E1 55.468} C_DIS
LIN {X 0.143,Y -287.333,Z 322.290,A 0.000,B 0.000,C 90.000,E1 52.110} C_DIS
LIN {X -0.177,Y -279.651,Z 322.275,A 0.000,B 0.000,C 90.000,E1 49.461} C_DIS
LIN {X -0.130,Y -273.834,Z 322.263,A 0.000,B 0.000,C 90.000,E1 47.391} C_DIS
LIN {X -0.066,Y -266.190,Z 322.248,A 0.000,B 0.000,C 90.000,E1 44.595} C_DIS
LIN {X 0.087,Y -260.612,Z 322.236,A 0.000,B 0.000,C 90.000,E1 42.447} C_DIS
LIN {X -0.145,Y -253.004,Z 322.220,A 0.000,B 0.000,C 90.000,E1 39.644} C_DIS
LIN {X -0.003,Y -247.263,Z 322.208,A 0.000,B 0.000,C 90.000,E1 37.443} C_DIS
LIN {X 0.070,Y -241.346,Z 322.196,A 0.000,B 0.000,C 90.000,E1 35.231} C_DIS
LIN {X -0.038,Y -233.528,Z 322.179,A 0.000,B 0.000,C 90.000,E1 32.291} C_DIS
LIN {X -0.059,Y -225.981,Z 322.163,A 0.000,B 0.000,C 90.000,E1 29.283} C_DIS
LIN {X -0.095,Y -218.990,Z 322.146,A 0.000,B 0.000,C 90.000,E1 26.232} C_DIS
LIN {X 0.087,Y -212.698,Z 322.128,A 0.000,B 0.000,C 90.000,E1 23.078} C_DIS
LIN {X 0.056,Y -207.310,Z 322.111,A 0.000,B 0.000,C 90.000,E1 19.939} C_DIS
LIN {X -0.112,Y -202.658,Z 322.093,A 0.000,B 0.000,C 90.000,E1 16.804} C_DIS
LIN {X -0.076,Y -197.849,Z 322.071,A 0.000,B 0.000,C 90.000,E1 12.771} C_DIS
LIN {X 0.015,Y -194.099,Z 322.048,A 0.000,B 0.000,C 90.000,E1 8.681} C_DIS
LIN {X 0.073,Y -190.654,Z 322.016,A 0.000,B 0.000,C 90.000,E1 2.922} C_DIS
LIN {X 0.058,Y -191.427,Z 321.929,A 0.000,B 0.000,C 90.000,E1 347.117} C_DIS
LIN {X 0.081,Y -194.795,Z 321.901,A 0.000,B 0.000,C 90.000,E1 342.181} C_DIS
LIN {X 0.085,Y -198.789,Z 321.878,A 0.000,B 0.000,C 90.000,E1 338.103} C_DIS
LIN {X 0.041,Y -203.774,Z 321.856,A 0.000,B 0.000,C 90.000,E1 334.076} C_DIS
LIN {X 0.058,Y -209.802,Z 321.834,A 0.000,B 0.000,C 90.000,E1 330.078} C_DIS
LIN {X -0.054,Y -216.697,Z 321.812,A 0.000,B 0.000,C 90.000,E1 326.167} C_DIS
LIN {X -0.030,Y -222.761,Z 321.795,A 0.000,B 0.000,C 90.000,E1 323.050} C_DIS
LIN {X -0.070,Y -229.522,Z 321.778,A 0.000,B 0.000,C 90.000,E1 319.989} C_DIS
LIN {X 0.002,Y -237.288,Z 321.761,A 0.000,B 0.000,C 90.000,E1 316.944} C_DIS
LIN {X 0.113,Y -246.198,Z 321.744,A 0.000,B 0.000,C 90.000,E1 313.947} C_DIS
LIN {X -0.025,Y -257.373,Z 321.726,A 0.000,B 0.000,C 90.000,E1 310.701} C_DIS
LIN {X -0.160,Y -269.422,Z 321.708,A 0.000,B 0.000,C 90.000,E1 307.523} C_DIS
LIN {X 0.055,Y -281.208,Z 321.693,A 0.000,B 0.000,C 90.000,E1 304.692} C_DIS
LIN {X -0.135,Y -294.262,Z 321.678,A 0.000,B 0.000,C 90.000,E1 302.005} C_DIS
LIN {X -0.061,Y -308.653,Z 321.663,A 0.000,B 0.000,C 90.000,E1 299.333} C_DIS
LIN {X 0.008,Y -322.471,Z 321.650,A 0.000,B 0.000,C 90.000,E1 297.052} C_DIS
LIN {X 0.059,Y -341.861,Z 321.635,A 0.000,B 0.000,C 90.000,E1 294.207} C_DIS
LIN {X 0.082,Y -362.047,Z 321.619,A 0.000,B 0.000,C 90.000,E1 291.461} C_DIS
LIN {X -0.089,Y -382.953,Z 321.605,A 0.000,B 0.000,C 90.000,E1 288.833} C_DIS
LIN {X -0.197,Y -399.969,Z 321.594,A 0.000,B 0.000,C 90.000,E1 286.858} C_DIS
LIN {X -0.132,Y -414.451,Z 321.584,A 0.000,B 0.000,C 90.000,E1 285.190} C_DIS
LIN {X -0.188,Y -426.547,Z 321.577,A 0.000,B 0.000,C 90.000,E1 283.828} C_DIS
LIN {X -0.106,Y -433.353,Z 321.572,A 0.000,B 0.000,C 90.000,E1 283.008} C_DIS
LIN {X 0.038,Y -439.645,Z 321.568,A 0.000,B 0.000,C 90.000,E1 282.187} C_DIS
LIN {X 0.036,Y -447.420,Z 321.562,A 0.000,B 0.000,C 90.000,E1 281.130} C_DIS
LIN {X 0.119,Y -454.601,Z 321.556,A 0.000,B 0.000,C 90.000,E1 280.074} C_DIS
LIN {X -0.041,Y -462.757,Z 321.549,A 0.000,B 0.000,C 90.000,E1 278.803} C_DIS
LIN {X -0.084,Y -470.264,Z 321.542,A 0.000,B 0.000,C 90.000,E1 277.530} C_DIS
LIN {X 0.184,Y -475.903,Z 321.536,A 0.000,B 0.000,C 90.000,E1 276.486} C_DIS
LIN {X 0.124,Y -479.671,Z 321.532,A 0.000,B 0.000,C 90.000,E1 275.739} C_DIS
LIN {X -0.066,Y -480.810,Z 321.531,A 0.000,B 0.000,C 90.000,E1 275.511} C_DIS
LIN {X 0.097,Y -482.725,Z 321.528,A 0.000,B 0.000,C 90.000,E1 274.992} C_DIS
LIN {X -0.219,Y -484.326,Z 321.525,A 0.000,B 0.000,C 90.000,E1 274.531} C_DIS
LIN {X -0.043,Y -485.464,Z 321.522,A 0.000,B 0.000,C 90.000,E1 274.012} C_DIS
LIN {X 0.109,Y -486.196,Z 321.520,A 0.000,B 0.000,C 90.000,E1 273.498} C_DIS
LIN {X -0.188,Y -486.591,Z 321.517,A 0.000,B 0.000,C 90.000,E1 273.037} C_DIS
LIN {X -0.020,Y -486.645,Z 321.514,A 0.000,B 0.000,C 90.000,E1 272.522} C_DIS
LIN {X -0.145,Y -486.150,Z 321.508,A 0.000,B 0.000,C 90.000,E1 271.547} C_DIS
LIN {X 0.199,Y -485.029,Z 321.503,A 0.000,B 0.000,C 90.000,E1 270.516} C_DIS
LIN {X -0.116,Y -484.066,Z 321.500,A 0.000,B 0.000,C 90.000,E1 270.057} C_DIS
LIN {X 0.049,Y -482.617,Z 321.497,A 0.000,B 0.000,C 90.000,E1 269.542} C_DIS
LIN {X 0.208,Y -480.635,Z 321.495,A 0.000,B 0.000,C 90.000,E1 269.026} C_DIS
LIN {X -0.124,Y -477.969,Z 321.492,A 0.000,B 0.000,C 90.000,E1 268.568} C_DIS
LIN {X 0.020,Y -474.425,Z 321.489,A 0.000,B 0.000,C 90.000,E1 268.051} C_DIS
LIN {X -0.160,Y -472.307,Z 321.488,A 0.000,B 0.000,C 90.000,E1 267.822} C_DIS
LIN {X -0.054,Y -467.165,Z 321.485,A 0.000,B 0.000,C 90.000,E1 267.306} C_DIS
LIN {X -0.237,Y -464.029,Z 321.484,A 0.000,B 0.000,C 90.000,E1 267.078} C_DIS
LIN {X -0.098,Y -460.981,Z 321.482,A 0.000,B 0.000,C 90.000,E1 266.846} C_DIS
LIN {X 0.014,Y -457.401,Z 321.481,A 0.000,B 0.000,C 90.000,E1 266.617} C_DIS
LIN {X 0.003,Y -454.040,Z 321.480,A 0.000,B 0.000,C 90.000,E1 266.445} C_DIS
LIN {X -0.142,Y -446.549,Z 321.479,A 0.000,B 0.000,C 90.000,E1 266.159} C_DIS
LIN {X -0.121,Y -438.702,Z 321.477,A 0.000,B 0.000,C 90.000,E1 265.927} C_DIS
LIN {X -0.073,Y -429.656,Z 321.476,A 0.000,B 0.000,C 90.000,E1 265.755} C_DIS
LIN {X 0.130,Y -420.552,Z 321.476,A 0.000,B 0.000,C 90.000,E1 265.641} C_DIS
LIN {X 0.055,Y -418.161,Z 321.476,A 0.000,B 0.000,C 90.000,E1 265.641} C_DIS
LIN {X -0.008,Y -180.909,Z 321.476,A 0.000,B 0.000,C 90.000,E1 265.641} C_DIS
LIN {X -0.078,Y -180.789,Z 321.471,A 0.000,B 0.000,C 90.000,E1 264.780} C_DIS
LIN {X -0.004,Y -178.887,Z 321.443,A 0.000,B 0.000,C 90.000,E1 259.690} C_DIS
LIN {X 0.071,Y -175.929,Z 321.414,A 0.000,B 0.000,C 90.000,E1 254.574} C_DIS
LIN {X 0.017,Y -175.372,Z 321.410,A 0.000,B 0.000,C 90.000,E1 253.740} C_DIS
LIN {X 0.075,Y -172.148,Z 321.386,A 0.000,B 0.000,C 90.000,E1 249.444} C_DIS
LIN {X 0.052,Y -171.613,Z 321.381,A 0.000,B 0.000,C 90.000,E1 248.592} C_DIS
LIN {X 0.040,Y -167.836,Z 321.357,A 0.000,B 0.000,C 90.000,E1 244.280} C_DIS
LIN {X 0.058,Y -166.564,Z 321.348,A 0.000,B 0.000,C 90.000,E1 242.538} C_DIS
LIN {X -0.033,Y -162.558,Z 321.323,A 0.000,B 0.000,C 90.000,E1 238.201} C_DIS
LIN {X 0.028,Y -161.236,Z 321.314,A 0.000,B 0.000,C 90.000,E1 236.421} C_DIS
LIN {X 0.062,Y -157.241,Z 321.289,A 0.000,B 0.000,C 90.000,E1 231.984} C_DIS
LIN {X -0.015,Y -155.964,Z 321.279,A 0.000,B 0.000,C 90.000,E1 230.231} C_DIS
LIN {X 0.042,Y -152.219,Z 321.254,A 0.000,B 0.000,C 90.000,E1 225.729} C_DIS
LIN {X 0.063,Y -150.462,Z 321.239,A 0.000,B 0.000,C 90.000,E1 223.014} C_DIS
LIN {X 0.089,Y -147.188,Z 321.214,A 0.000,B 0.000,C 90.000,E1 218.463} C_DIS
LIN {X 0.056,Y -145.206,Z 321.194,A 0.000,B 0.000,C 90.000,E1 214.818} C_DIS
LIN {X -0.035,Y -142.341,Z 321.163,A 0.000,B 0.000,C 90.000,E1 209.333} C_DIS
LIN {X 0.019,Y -141.729,Z 321.153,A 0.000,B 0.000,C 90.000,E1 207.462} C_DIS
LIN {X 0.001,Y -139.482,Z 321.117,A 0.000,B 0.000,C 90.000,E1 200.972} C_DIS
LIN {X -0.010,Y -138.981,Z 321.101,A 0.000,B 0.000,C 90.000,E1 198.181} C_DIS
LIN {X -0.050,Y -138.333,Z 321.054,A 0.000,B 0.000,C 90.000,E1 189.792} C_DIS
LIN {X -0.025,Y -139.428,Z 321.008,A 0.000,B 0.000,C 90.000,E1 181.375} C_DIS
LIN {X 0.028,Y -141.353,Z 320.971,A 0.000,B 0.000,C 90.000,E1 174.837} C_DIS
LIN {X 0.005,Y -142.707,Z 320.956,A 0.000,B 0.000,C 90.000,E1 172.064} C_DIS
LIN {X -0.036,Y -145.080,Z 320.930,A 0.000,B 0.000,C 90.000,E1 167.465} C_DIS
LIN {X -0.040,Y -147.705,Z 320.910,A 0.000,B 0.000,C 90.000,E1 163.795} C_DIS
LIN {X 0.043,Y -150.358,Z 320.890,A 0.000,B 0.000,C 90.000,E1 160.115} C_DIS
LIN {X 0.062,Y -153.783,Z 320.869,A 0.000,B 0.000,C 90.000,E1 156.485} C_DIS
LIN {X -0.018,Y -157.195,Z 320.850,A 0.000,B 0.000,C 90.000,E1 152.922} C_DIS
LIN {X 0.064,Y -161.356,Z 320.830,A 0.000,B 0.000,C 90.000,E1 149.331} C_DIS
LIN {X 0.076,Y -165.559,Z 320.810,A 0.000,B 0.000,C 90.000,E1 145.801} C_DIS
LIN {X -0.041,Y -170.475,Z 320.791,A 0.000,B 0.000,C 90.000,E1 142.351} C_DIS
LIN {X 0.109,Y -175.357,Z 320.772,A 0.000,B 0.000,C 90.000,E1 138.852} C_DIS
LIN {X -0.028,Y -180.980,Z 320.753,A 0.000,B 0.000,C 90.000,E1 135.486} C_DIS
LIN {X -0.041,Y -186.405,Z 320.734,A 0.000,B 0.000,C 90.000,E1 132.123} C_DIS
LIN {X -0.101,Y -191.034,Z 320.720,A 0.000,B 0.000,C 90.000,E1 129.644} C_DIS
LIN {X 0.090,Y -196.816,Z 320.702,A 0.000,B 0.000,C 90.000,E1 126.297} C_DIS
LIN {X 0.009,Y -200.070,Z 320.693,A 0.000,B 0.000,C 90.000,E1 124.692} C_DIS
LIN {X -0.024,Y -201.656,Z 320.688,A 0.000,B 0.000,C 90.000,E1 123.833} C_DIS
LIN {X -0.090,Y -303.114,Z 320.688,A 0.000,B 0.000,C 90.000,E1 123.833} C_DIS
LIN {X 0.025,Y -308.262,Z 320.687,A 0.000,B 0.000,C 90.000,E1 123.627} C_DIS
LIN {X -0.029,Y -310.731,Z 320.686,A 0.000,B 0.000,C 90.000,E1 123.452} C_DIS
LIN {X -0.054,Y -314.048,Z 320.684,A 0.000,B 0.000,C 90.000,E1 123.086} C_DIS
LIN {X 0.106,Y -316.006,Z 320.682,A 0.000,B 0.000,C 90.000,E1 122.752} C_DIS
LIN {X 0.001,Y -317.545,Z 320.680,A 0.000,B 0.000,C 90.000,E1 122.467} C_DIS
LIN {X 0.023,Y -322.297,Z 320.673,A 0.000,B 0.000,C 90.000,E1 121.180} C_DIS
LIN {X -0.130,Y -333.580,Z 320.657,A 0.000,B 0.000,C 90.000,E1 118.359} C_DIS
LIN {X 0.032,Y -346.297,Z 320.642,A 0.000,B 0.000,C 90.000,E1 115.540} C_DIS
LIN {X -0.102,Y -358.894,Z 320.628,A 0.000,B 0.000,C 90.000,E1 113.131} C_DIS
LIN {X -0.013,Y -372.805,Z 320.615,A 0.000,B 0.000,C 90.000,E1 110.737} C_DIS
LIN {X -0.049,Y -388.132,Z 320.602,A 0.000,B 0.000,C 90.000,E1 108.417} C_DIS
LIN {X 0.044,Y -404.989,Z 320.590,A 0.000,B 0.000,C 90.000,E1 106.134} C_DIS
LIN {X -0.065,Y -423.501,Z 320.577,A 0.000,B 0.000,C 90.000,E1 103.939} C_DIS
LIN {X -0.058,Y -443.431,Z 320.566,A 0.000,B 0.000,C 90.000,E1 101.827} C_DIS
LIN {X -0.183,Y -463.961,Z 320.555,A 0.000,B 0.000,C 90.000,E1 99.905} C_DIS
LIN {X 0.211,Y -487.640,Z 320.544,A 0.000,B 0.000,C 90.000,E1 97.871} C_DIS
LIN {X -0.195,Y -495.632,Z 320.540,A 0.000,B 0.000,C 90.000,E1 97.296} C_DIS
LIN {X 0.229,Y -499.378,Z 320.538,A 0.000,B 0.000,C 90.000,E1 96.834} C_DIS
LIN {X 0.082,Y -500.857,Z 320.537,A 0.000,B 0.000,C 90.000,E1 96.606} C_DIS
LIN {X -0.008,Y -501.957,Z 320.535,A 0.000,B 0.000,C 90.000,E1 96.372} C_DIS
LIN {X -0.218,Y -503.236,Z 320.533,A 0.000,B 0.000,C 90.000,E1 95.910} C_DIS
LIN {X 0.077,Y -503.475,Z 320.530,A 0.000,B 0.000,C 90.000,E1 95.391} C_DIS
LIN {X -0.165,Y -502.707,Z 320.527,A 0.000,B 0.000,C 90.000,E1 94.935} C_DIS
LIN {X 0.139,Y -500.800,Z 320.525,A 0.000,B 0.000,C 90.000,E1 94.416} C_DIS
LIN {X -0.064,Y -497.564,Z 320.522,A 0.000,B 0.000,C 90.000,E1 93.955} C_DIS
LIN {X -0.065,Y -489.937,Z 320.517,A 0.000,B 0.000,C 90.000,E1 92.980} C_DIS
LIN {X 0.003,Y -477.640,Z 320.508,A 0.000,B 0.000,C 90.000,E1 91.489} C_DIS
LIN {X -0.045,Y -457.755,Z 320.494,A 0.000,B 0.000,C 90.000,E1 88.969} C_DIS
LIN {X 0.101,Y -441.441,Z 320.481,A 0.000,B 0.000,C 90.000,E1 86.617} C_DIS
LIN {X -0.131,Y -426.454,Z 320.468,A 0.000,B 0.000,C 90.000,E1 84.261} C_DIS
LIN {X 0.186,Y -406.927,Z 320.448,A 0.000,B 0.000,C 90.000,E1 80.679} C_DIS
LIN {X 0.002,Y -396.924,Z 320.438,A 0.000,B 0.000,C 90.000,E1 78.757} C_DIS
LIN {X 0.158,Y -386.774,Z 320.427,A 0.000,B 0.000,C 90.000,E1 76.756} C_DIS
LIN {X -0.139,Y -373.742,Z 320.412,A 0.000,B 0.000,C 90.000,E1 74.212} C_DIS
LIN {X 0.081,Y -363.594,Z 320.401,A 0.000,B 0.000,C 90.000,E1 72.127} C_DIS
LIN {X -0.093,Y -354.863,Z 320.391,A 0.000,B 0.000,C 90.000,E1 70.369} C_DIS
LIN {X 0.091,Y -341.861,Z 320.376,A 0.000,B 0.000,C 90.000,E1 67.614} C_DIS
LIN {X 0.022,Y -331.323,Z 320.362,A 0.000,B 0.000,C 90.000,E1 65.153} C_DIS
LIN {X -0.110,Y -319.430,Z 320.344,A 0.000,B 0.000,C 90.000,E1 62.025} C_DIS
LIN {X -0.059,Y -309.274,Z 320.328,A 0.000,B 0.000,C 90.000,E1 59.125} C_DIS
LIN {X -0.006,Y -297.558,Z 320.308,A 0.000,B 0.000,C 90.000,E1 55.515} C_DIS
LIN {X -0.060,Y -287.671,Z 320.290,A 0.000,B 0.000,C 90.000,E1 52.190} C_DIS
LIN {X 0.027,Y -279.967,Z 320.275,A 0.000,B 0.000,C 90.000,E1 49.461} C_DIS
LIN {X 0.065,Y -272.190,Z 320.260,A 0.000,B 0.000,C 90.000,E1 46.701} C_DIS
LIN {X -0.108,Y -264.606,Z 320.244,A 0.000,B 0.000,C 90.000,E1 43.947} C_DIS
LIN {X -0.162,Y -259.018,Z 320.232,A 0.000,B 0.000,C 90.000,E1 41.838} C_DIS
LIN {X 0.124,Y -251.431,Z 320.216,A 0.000,B 0.000,C 90.000,E1 38.910} C_DIS
LIN {X 0.080,Y -245.653,Z 320.204,A 0.000,B 0.000,C 90.000,E1 36.744} C_DIS
LIN {X -0.047,Y -237.723,Z 320.188,A 0.000,B 0.000,C 90.000,E1 33.833} C_DIS
LIN {X -0.049,Y -230.049,Z 320.171,A 0.000,B 0.000,C 90.000,E1 30.846} C_DIS
LIN {X 0.112,Y -222.665,Z 320.154,A 0.000,B 0.000,C 90.000,E1 27.769} C_DIS
LIN {X -0.012,Y -215.995,Z 320.137,A 0.000,B 0.000,C 90.000,E1 24.719} C_DIS
LIN {X 0.008,Y -210.168,Z 320.120,A 0.000,B 0.000,C 90.000,E1 21.589} C_DIS
LIN {X 0.038,Y -205.129,Z 320.102,A 0.000,B 0.000,C 90.000,E1 18.417} C_DIS
LIN {X -0.054,Y -200.877,Z 320.085,A 0.000,B 0.000,C 90.000,E1 15.245} C_DIS
LIN {X 0.018,Y -196.443,Z 320.062,A 0.000,B 0.000,C 90.000,E1 11.186} C_DIS
LIN {X -0.031,Y -193.161,Z 320.040,A 0.000,B 0.000,C 90.000,E1 7.125} C_DIS
LIN {X -0.034,Y -190.259,Z 320.008,A 0.000,B 0.000,C 90.000,E1 1.375} C_DIS
LIN {X 0.071,Y -191.548,Z 319.929,A 0.000,B 0.000,C 90.000,E1 347.117} C_DIS
LIN {X 0.098,Y -194.905,Z 319.901,A 0.000,B 0.000,C 90.000,E1 342.181} C_DIS
LIN {X -0.079,Y -198.870,Z 319.879,A 0.000,B 0.000,C 90.000,E1 338.156} C_DIS
LIN {X -0.024,Y -203.839,Z 319.856,A 0.000,B 0.000,C 90.000,E1 334.101} C_DIS
LIN {X -0.097,Y -209.869,Z 319.834,A 0.000,B 0.000,C 90.000,E1 330.127} C_DIS
LIN {X -0.025,Y -216.720,Z 319.812,A 0.000,B 0.000,C 90.000,E1 326.167} C_DIS
LIN {X 0.000,Y -222.781,Z 319.795,A 0.000,B 0.000,C 90.000,E1 323.050} C_DIS
LIN {X -0.038,Y -229.552,Z 319.778,A 0.000,B 0.000,C 90.000,E1 319.989} C_DIS
LIN {X 0.042,Y -237.335,Z 319.761,A 0.000,B 0.000,C 90.000,E1 316.944} C_DIS
LIN {X 0.156,Y -246.266,Z 319.744,A 0.000,B 0.000,C 90.000,E1 313.947} C_DIS
LIN {X 0.022,Y -257.466,Z 319.726,A 0.000,B 0.000,C 90.000,E1 310.701} C_DIS
LIN {X -0.108,Y -269.545,Z 319.708,A 0.000,B 0.000,C 90.000,E1 307.523} C_DIS
LIN {X 0.113,Y -281.368,Z 319.693,A 0.000,B 0.000,C 90.000,E1 304.692} C_DIS
LIN {X -0.070,Y -294.426,Z 319.678,A 0.000,B 0.000,C 90.000,E1 302.005} C_DIS
LIN {X 0.011,Y -308.861,Z 319.663,A 0.000,B 0.000,C 90.000,E1 299.333} C_DIS
LIN {X -0.057,Y -322.732,Z 319.650,A 0.000,B 0.000,C 90.000,E1 297.078} C_DIS
LIN {X 0.152,Y -342.130,Z 319.635,A 0.000,B 0.000,C 90.000,E1 294.207} C_DIS
LIN {X 0.132,Y -360.029,Z 319.621,A 0.000,B 0.000,C 90.000,E1 291.770} C_DIS
LIN {X 0.160,Y -378.408,Z 319.608,A 0.000,B 0.000,C 90.000,E1 289.396} C_DIS
LIN {X 0.213,Y -397.703,Z 319.595,A 0.000,B 0.000,C 90.000,E1 287.094} C_DIS
LIN {X 0.128,Y -412.269,Z 319.586,A 0.000,B 0.000,C 90.000,E1 285.426} C_DIS
LIN {X 0.053,Y -424.338,Z 319.578,A 0.000,B 0.000,C 90.000,E1 284.064} C_DIS
LIN {X 0.111,Y -431.266,Z 319.574,A 0.000,B 0.000,C 90.000,E1 283.244} C_DIS
LIN {X -0.182,Y -437.702,Z 319.569,A 0.000,B 0.000,C 90.000,E1 282.479} C_DIS
LIN {X -0.211,Y -445.587,Z 319.563,A 0.000,B 0.000,C 90.000,E1 281.422} C_DIS
LIN {X -0.152,Y -452.875,Z 319.557,A 0.000,B 0.000,C 90.000,E1 280.366} C_DIS
LIN {X -0.090,Y -459.535,Z 319.552,A 0.000,B 0.000,C 90.000,E1 279.321} C_DIS
LIN {X 0.051,Y -465.754,Z 319.546,A 0.000,B 0.000,C 90.000,E1 278.276} C_DIS
LIN {X 0.046,Y -473.051,Z 319.539,A 0.000,B 0.000,C 90.000,E1 277.004} C_DIS
LIN {X -0.189,Y -478.349,Z 319.533,A 0.000,B 0.000,C 90.000,E1 276.024} C_DIS
LIN {X -0.092,Y -480.679,Z 319.531,A 0.000,B 0.000,C 90.000,E1 275.511} C_DIS
LIN {X 0.069,Y -482.609,Z 319.528,A 0.000,B 0.000,C 90.000,E1 274.992} C_DIS
LIN {X 0.235,Y -484.161,Z 319.525,A 0.000,B 0.000,C 90.000,E1 274.473} C_DIS
LIN {X -0.073,Y -485.346,Z 319.522,A 0.000,B 0.000,C 90.000,E1 274.012} C_DIS
LIN {X 0.078,Y -486.116,Z 319.519,A 0.000,B 0.000,C 90.000,E1 273.498} C_DIS
LIN {X -0.219,Y -486.492,Z 319.517,A 0.000,B 0.000,C 90.000,E1 273.037} C_DIS
LIN {X -0.053,Y -486.564,Z 319.514,A 0.000,B 0.000,C 90.000,E1 272.522} C_DIS
LIN {X 0.119,Y -486.401,Z 319.511,A 0.000,B 0.000,C 90.000,E1 272.007} C_DIS
LIN {X -0.006,Y -485.544,Z 319.506,A 0.000,B 0.000,C 90.000,E1 271.031} C_DIS
LIN {X 0.165,Y -484.888,Z 319.503,A 0.000,B 0.000,C 90.000,E1 270.516} C_DIS
LIN {X -0.151,Y -483.927,Z 319.500,A 0.000,B 0.000,C 90.000,E1 270.057} C_DIS
LIN {X 0.014,Y -482.499,Z 319.497,A 0.000,B 0.000,C 90.000,E1 269.542} C_DIS
LIN {X 0.172,Y -480.517,Z 319.495,A 0.000,B 0.000,C 90.000,E1 269.026} C_DIS
LIN {X 0.005,Y -479.319,Z 319.493,A 0.000,B 0.000,C 90.000,E1 268.797} C_DIS
LIN {X 0.142,Y -476.244,Z 319.491,A 0.000,B 0.000,C 90.000,E1 268.282} C_DIS
LIN {X -0.196,Y -472.268,Z 319.488,A 0.000,B 0.000,C 90.000,E1 267.822} C_DIS
LIN {X 0.094,Y -469.877,Z 319.486,A 0.000,B 0.000,C 90.000,E1 267.535} C_DIS
LIN {X -0.097,Y -467.174,Z 319.485,A 0.000,B 0.000,C 90.000,E1 267.306} C_DIS
LIN {X 0.176,Y -464.073,Z 319.484,A 0.000,B 0.000,C 90.000,E1 267.020} C_DIS
LIN {X -0.168,Y -461.021,Z 319.482,A 0.000,B 0.000,C 90.000,E1 266.846} C_DIS
LIN {X -0.073,Y -457.482,Z 319.481,A 0.000,B 0.000,C 90.000,E1 266.617} C_DIS
LIN {X -0.144,Y -449.974,Z 319.479,A 0.000,B 0.000,C 90.000,E1 266.274} C_DIS
LIN {X 0.020,Y -442.253,Z 319.478,A 0.000,B 0.000,C 90.000,E1 265.988} C_DIS
LIN {X -0.140,Y -433.670,Z 319.477,A 0.000,B 0.000,C 90.000,E1 265.812} C_DIS
LIN {X -0.196,Y -429.579,Z 319.476,A 0.000,B 0.000,C 90.000,E1 265.755} C_DIS
LIN {X 0.027,Y -420.076,Z 319.476,A 0.000,B 0.000,C 90.000,E1 265.641} C_DIS
LIN {X -0.044,Y -417.713,Z 319.476,A 0.000,B 0.000,C 90.000,E1 265.641} C_DIS
LIN {X -0.050,Y -180.909,Z 319.476,A 0.000,B 0.000,C 90.000,E1 265.641} C_DIS
LIN {X 0.064,Y -180.784,Z 319.471,A 0.000,B 0.000,C 90.000,E1 264.723} C_DIS
LIN {X -0.041,Y -178.882,Z 319.443,A 0.000,B 0.000,C 90.000,E1 259.690} C_DIS
LIN {X 0.035,Y -175.924,Z 319.414,A 0.000,B 0.000,C 90.000,E1 254.574} C_DIS
LIN {X -0.019,Y -175.362,Z 319.410,A 0.000,B 0.000,C 90.000,E1 253.740} C_DIS
LIN {X 0.039,Y -172.141,Z 319.386,A 0.000,B 0.000,C 90.000,E1 249.444} C_DIS
LIN {X 0.016,Y -171.605,Z 319.381,A 0.000,B 0.000,C 90.000,E1 248.592} C_DIS
LIN {X 0.005,Y -167.827,Z 319.357,A 0.000,B 0.000,C 90.000,E1 244.280} C_DIS
LIN {X 0.022,Y -166.552,Z 319.347,A 0.000,B 0.000,C 90.000,E1 242.538} C_DIS
LIN {X -0.067,Y -162.547,Z 319.323,A 0.000,B 0.000,C 90.000,E1 238.201} C_DIS
LIN {X -0.007,Y -161.225,Z 319.313,A 0.000,B 0.000,C 90.000,E1 236.421} C_DIS
LIN {X 0.028,Y -157.231,Z 319.289,A 0.000,B 0.000,C 90.000,E1 231.984} C_DIS
LIN {X 0.050,Y -155.956,Z 319.279,A 0.000,B 0.000,C 90.000,E1 230.194} C_DIS
LIN {X 0.009,Y -152.209,Z 319.254,A 0.000,B 0.000,C 90.000,E1 225.729} C_DIS
LIN {X 0.030,Y -150.454,Z 319.239,A 0.000,B 0.000,C 90.000,E1 223.014} C_DIS
LIN {X 0.056,Y -147.179,Z 319.214,A 0.000,B 0.000,C 90.000,E1 218.463} C_DIS
LIN {X 0.023,Y -145.197,Z 319.193,A 0.000,B 0.000,C 90.000,E1 214.818} C_DIS
LIN {X 0.058,Y -142.337,Z 319.163,A 0.000,B 0.000,C 90.000,E1 209.283} C_DIS
LIN {X -0.013,Y -141.725,Z 319.153,A 0.000,B 0.000,C 90.000,E1 207.462} C_DIS
LIN {X -0.031,Y -139.480,Z 319.116,A 0.000,B 0.000,C 90.000,E1 200.972} C_DIS
LIN {X -0.042,Y -138.977,Z 319.101,A 0.000,B 0.000,C 90.000,E1 198.181} C_DIS
LIN {X 0.079,Y -138.332,Z 319.054,A 0.000,B 0.000,C 90.000,E1 189.726} C_DIS
LIN {X -0.057,Y -139.431,Z 319.008,A 0.000,B 0.000,C 90.000,E1 181.375} C_DIS
LIN {X 0.022,Y -140.956,Z 318.976,A 0.000,B 0.000,C 90.000,E1 175.755} C_DIS
LIN {X -0.028,Y -142.712,Z 318.956,A 0.000,B 0.000,C 90.000,E1 172.064} C_DIS
LIN {X -0.069,Y -145.088,Z 318.930,A 0.000,B 0.000,C 90.000,E1 167.465} C_DIS
LIN {X 0.068,Y -147.713,Z 318.910,A 0.000,B 0.000,C 90.000,E1 163.740} C_DIS
LIN {X 0.010,Y -150.369,Z 318.890,A 0.000,B 0.000,C 90.000,E1 160.115} C_DIS
LIN {X 0.027,Y -153.797,Z 318.869,A 0.000,B 0.000,C 90.000,E1 156.485} C_DIS
LIN {X -0.053,Y -157.209,Z 318.849,A 0.000,B 0.000,C 90.000,E1 152.922} C_DIS
LIN {X 0.029,Y -161.372,Z 318.830,A 0.000,B 0.000,C 90.000,E1 149.331} C_DIS
LIN {X 0.040,Y -165.574,Z 318.810,A 0.000,B 0.000,C 90.000,E1 145.801} C_DIS
LIN {X 0.028,Y -170.494,Z 318.791,A 0.000,B 0.000,C 90.000,E1 142.316} C_DIS
LIN {X 0.072,Y -175.374,Z 318.772,A 0.000,B 0.000,C 90.000,E1 138.852} C_DIS
LIN {X -0.065,Y -180.998,Z 318.753,A 0.000,B 0.000,C 90.000,E1 135.486} C_DIS
LIN {X 0.059,Y -186.426,Z 318.734,A 0.000,B 0.000,C 90.000,E1 132.081} C_DIS
LIN {X 0.007,Y -191.053,Z 318.720,A 0.000,B 0.000,C 90.000,E1 129.600} C_DIS
LIN {X 0.051,Y -196.838,Z 318.702,A 0.000,B 0.000,C 90.000,E1 126.297} C_DIS
LIN {X -0.030,Y -200.094,Z 318.693,A 0.000,B 0.000,C 90.000,E1 124.692} C_DIS
LIN {X -0.027,Y -201.740,Z 318.688,A 0.000,B 0.000,C 90.000,E1 123.785} C_DIS
LIN {X -0.093,Y -302.782,Z 318.688,A 0.000,B 0.000,C 90.000,E1 123.785} C_DIS
LIN {X 0.171,Y -304.682,Z 318.687,A 0.000,B 0.000,C 90.000,E1 123.706} C_DIS
LIN {X -0.048,Y -308.563,Z 318.686,A 0.000,B 0.000,C 90.000,E1 123.579} C_DIS
LIN {X -0.100,Y -310.804,Z 318.686,A 0.000,B 0.000,C 90.000,E1 123.420} C_DIS
LIN {X -0.115,Y -313.904,Z 318.684,A 0.000,B 0.000,C 90.000,E1 123.086} C_DIS
LIN {X 0.077,Y -315.901,Z 318.682,A 0.000,B 0.000,C 90.000,E1 122.752} C_DIS
LIN {X 0.004,Y -317.467,Z 318.680,A 0.000,B 0.000,C 90.000,E1 122.467} C_DIS
LIN {X 0.141,Y -319.949,Z 318.677,A 0.000,B 0.000,C 90.000,E1 121.799} C_DIS
LIN {X 0.093,Y -330.929,Z 318.661,A 0.000,B 0.000,C 90.000,E1 118.949} C_DIS
LIN {X 0.031,Y -343.317,Z 318.645,A 0.000,B 0.000,C 90.000,E1 116.155} C_DIS
LIN {X 0.141,Y -355.600,Z 318.632,A 0.000,B 0.000,C 90.000,E1 113.695} C_DIS
LIN {X -0.054,Y -369.175,Z 318.618,A 0.000,B 0.000,C 90.000,E1 111.334} C_DIS
LIN {X 0.170,Y -384.137,Z 318.605,A 0.000,B 0.000,C 90.000,E1 108.960} C_DIS
LIN {X 0.174,Y -400.601,Z 318.593,A 0.000,B 0.000,C 90.000,E1 106.677} C_DIS
LIN {X -0.030,Y -418.686,Z 318.580,A 0.000,B 0.000,C 90.000,E1 104.481} C_DIS
LIN {X -0.190,Y -438.360,Z 318.569,A 0.000,B 0.000,C 90.000,E1 102.355} C_DIS
LIN {X -0.127,Y -458.754,Z 318.557,A 0.000,B 0.000,C 90.000,E1 100.366} C_DIS
LIN {X -0.171,Y -482.300,Z 318.546,A 0.000,B 0.000,C 90.000,E1 98.341} C_DIS
LIN {X -0.200,Y -495.628,Z 318.540,A 0.000,B 0.000,C 90.000,E1 97.296} C_DIS
LIN {X 0.243,Y -499.452,Z 318.538,A 0.000,B 0.000,C 90.000,E1 96.834} C_DIS
LIN {X 0.096,Y -500.968,Z 318.537,A 0.000,B 0.000,C 90.000,E1 96.606} C_DIS
LIN {X 0.006,Y -502.099,Z 318.535,A 0.000,B 0.000,C 90.000,E1 96.372} C_DIS
LIN {X -0.203,Y -503.431,Z 318.533,A 0.000,B 0.000,C 90.000,E1 95.910} C_DIS
LIN {X 0.093,Y -503.716,Z 318.530,A 0.000,B 0.000,C 90.000,E1 95.391} C_DIS
LIN {X -0.149,Y -502.996,Z 318.527,A 0.000,B 0.000,C 90.000,E1 94.935} C_DIS
LIN {X 0.157,Y -501.145,Z 318.525,A 0.000,B 0.000,C 90.000,E1 94.416} C_DIS
LIN {X 0.038,Y -499.680,Z 318.523,A 0.000,B 0.000,C 90.000,E1 94.188} C_DIS
LIN {X 0.065,Y -492.290,Z 318.518,A 0.000,B 0.000,C 90.000,E1 93.212} C_DIS
LIN {X -0.141,Y -482.138,Z 318.511,A 0.000,B 0.000,C 90.000,E1 92.007} C_DIS
LIN {X -0.007,Y -458.067,Z 318.494,A 0.000,B 0.000,C 90.000,E1 88.969} C_DIS
LIN {X 0.145,Y -441.734,Z 318.481,A 0.000,B 0.000,C 90.000,E1 86.617} C_DIS
LIN {X -0.081,Y -426.718,Z 318.468,A 0.000,B 0.000,C 90.000,E1 84.261} C_DIS
LIN {X -0.159,Y -407.200,Z 318.448,A 0.000,B 0.000,C 90.000,E1 80.735} C_DIS
LIN {X 0.063,Y -397.199,Z 318.438,A 0.000,B 0.000,C 90.000,E1 78.757} C_DIS
LIN {X 0.135,Y -387.038,Z 318.427,A 0.000,B 0.000,C 90.000,E1 76.769} C_DIS
LIN {X -0.069,Y -374.030,Z 318.412,A 0.000,B 0.000,C 90.000,E1 74.212} C_DIS
LIN {X 0.155,Y -363.877,Z 318.401,A 0.000,B 0.000,C 90.000,E1 72.127} C_DIS
LIN {X -0.015,Y -355.158,Z 318.391,A 0.000,B 0.000,C 90.000,E1 70.369} C_DIS
LIN {X -0.164,Y -343.566,Z 318.378,A 0.000,B 0.000,C 90.000,E1 67.975} C_DIS
LIN {X -0.013,Y -332.869,Z 318.364,A 0.000,B 0.000,C 90.000,E1 65.485} C_DIS
LIN {X -0.017,Y -319.747,Z 318.345,A 0.000,B 0.000,C 90.000,E1 62.025} C_DIS
LIN {X 0.041,Y -309.596,Z 318.329,A 0.000,B 0.000,C 90.000,E1 59.125} C_DIS
LIN {X 0.100,Y -297.859,Z 318.309,A 0.000,B 0.000,C 90.000,E1 55.515} C_DIS
LIN {X 0.051,Y -287.941,Z 318.290,A 0.000,B 0.000,C 90.000,E1 52.190} C_DIS
LIN {X -0.114,Y -282.151,Z 318.279,A 0.000,B 0.000,C 90.000,E1 50.194} C_DIS
LIN {X 0.004,Y -276.321,Z 318.267,A 0.000,B 0.000,C 90.000,E1 48.119} C_DIS
LIN {X 0.119,Y -268.597,Z 318.252,A 0.000,B 0.000,C 90.000,E1 45.324} C_DIS
LIN {X 0.048,Y -261.135,Z 318.236,A 0.000,B 0.000,C 90.000,E1 42.528} C_DIS
LIN {X -0.049,Y -255.446,Z 318.224,A 0.000,B 0.000,C 90.000,E1 40.415} C_DIS
LIN {X -0.054,Y -249.775,Z 318.212,A 0.000,B 0.000,C 90.000,E1 38.257} C_DIS
LIN {X -0.123,Y -243.953,Z 318.200,A 0.000,B 0.000,C 90.000,E1 36.091} C_DIS
LIN {X 0.100,Y -236.031,Z 318.184,A 0.000,B 0.000,C 90.000,E1 33.086} C_DIS
LIN {X -0.065,Y -228.387,Z 318.167,A 0.000,B 0.000,C 90.000,E1 30.129} C_DIS
LIN {X -0.044,Y -221.149,Z 318.150,A 0.000,B 0.000,C 90.000,E1 27.078} C_DIS
LIN {X 0.090,Y -214.673,Z 318.133,A 0.000,B 0.000,C 90.000,E1 23.951} C_DIS
LIN {X -0.011,Y -209.081,Z 318.116,A 0.000,B 0.000,C 90.000,E1 20.844} C_DIS
LIN {X -0.079,Y -204.195,Z 318.098,A 0.000,B 0.000,C 90.000,E1 17.692} C_DIS
LIN {X 0.047,Y -199.217,Z 318.076,A 0.000,B 0.000,C 90.000,E1 13.647} C_DIS
LIN {X -0.014,Y -195.208,Z 318.053,A 0.000,B 0.000,C 90.000,E1 9.613} C_DIS
LIN {X 0.001,Y -191.856,Z 318.026,A 0.000,B 0.000,C 90.000,E1 4.702} C_DIS
LIN {X -0.079,Y -189.519,Z 317.984,A 0.000,B 0.000,C 90.000,E1 357.078} C_DIS
LIN {X -0.090,Y -191.247,Z 317.933,A 0.000,B 0.000,C 90.000,E1 347.993} C_DIS
LIN {X 0.063,Y -194.359,Z 317.906,A 0.000,B 0.000,C 90.000,E1 343.015} C_DIS
LIN {X -0.008,Y -198.086,Z 317.883,A 0.000,B 0.000,C 90.000,E1 338.954} C_DIS
LIN {X -0.054,Y -202.833,Z 317.861,A 0.000,B 0.000,C 90.000,E1 334.921} C_DIS
LIN {X -0.074,Y -208.650,Z 317.838,A 0.000,B 0.000,C 90.000,E1 330.923} C_DIS
LIN {X -0.037,Y -215.331,Z 317.816,A 0.000,B 0.000,C 90.000,E1 326.962} C_DIS
LIN {X 0.011,Y -221.214,Z 317.799,A 0.000,B 0.000,C 90.000,E1 323.829} C_DIS
LIN {X 0.116,Y -227.797,Z 317.782,A 0.000,B 0.000,C 90.000,E1 320.723} C_DIS
LIN {X -0.004,Y -235.344,Z 317.765,A 0.000,B 0.000,C 90.000,E1 317.715} C_DIS
LIN {X -0.115,Y -244.030,Z 317.749,A 0.000,B 0.000,C 90.000,E1 314.757} C_DIS
LIN {X 0.017,Y -254.997,Z 317.730,A 0.000,B 0.000,C 90.000,E1 311.434} C_DIS
LIN {X -0.024,Y -266.893,Z 317.712,A 0.000,B 0.000,C 90.000,E1 308.222} C_DIS
LIN {X -0.163,Y -279.976,Z 317.695,A 0.000,B 0.000,C 90.000,E1 305.105} C_DIS
LIN {X 0.008,Y -292.877,Z 317.680,A 0.000,B 0.000,C 90.000,E1 302.339} C_DIS
LIN {X 0.082,Y -309.090,Z 317.663,A 0.000,B 0.000,C 90.000,E1 299.333} C_DIS
LIN {X 0.093,Y -320.925,Z 317.652,A 0.000,B 0.000,C 90.000,E1 297.385} C_DIS
LIN {X -0.052,Y -340.204,Z 317.636,A 0.000,B 0.000,C 90.000,E1 294.567} C_DIS
LIN {X 0.101,Y -360.297,Z 317.621,A 0.000,B 0.000,C 90.000,E1 291.791} C_DIS
LIN {X -0.082,Y -378.611,Z 317.608,A 0.000,B 0.000,C 90.000,E1 289.450} C_DIS
LIN {X -0.089,Y -397.885,Z 317.595,A 0.000,B 0.000,C 90.000,E1 287.149} C_DIS
LIN {X 0.211,Y -412.388,Z 317.586,A 0.000,B 0.000,C 90.000,E1 285.426} C_DIS
LIN {X 0.141,Y -424.399,Z 317.578,A 0.000,B 0.000,C 90.000,E1 284.064} C_DIS
LIN {X -0.040,Y -433.480,Z 317.572,A 0.000,B 0.000,C 90.000,E1 283.008} C_DIS
LIN {X 0.106,Y -439.689,Z 317.568,A 0.000,B 0.000,C 90.000,E1 282.187} C_DIS
LIN {X 0.106,Y -447.413,Z 317.562,A 0.000,B 0.000,C 90.000,E1 281.130} C_DIS
LIN {X 0.190,Y -454.502,Z 317.556,A 0.000,B 0.000,C 90.000,E1 280.074} C_DIS
LIN {X 0.030,Y -462.576,Z 317.549,A 0.000,B 0.000,C 90.000,E1 278.803} C_DIS
LIN {X 0.211,Y -468.544,Z 317.543,A 0.000,B 0.000,C 90.000,E1 277.757} C_DIS
LIN {X -0.068,Y -474.244,Z 317.538,A 0.000,B 0.000,C 90.000,E1 276.777} C_DIS
LIN {X 0.189,Y -479.344,Z 317.532,A 0.000,B 0.000,C 90.000,E1 275.739} C_DIS
LIN {X -0.001,Y -480.486,Z 317.531,A 0.000,B 0.000,C 90.000,E1 275.511} C_DIS
LIN {X 0.159,Y -482.450,Z 317.528,A 0.000,B 0.000,C 90.000,E1 274.992} C_DIS
LIN {X -0.158,Y -484.024,Z 317.525,A 0.000,B 0.000,C 90.000,E1 274.531} C_DIS
LIN {X 0.016,Y -485.217,Z 317.522,A 0.000,B 0.000,C 90.000,E1 274.012} C_DIS
LIN {X 0.166,Y -485.980,Z 317.520,A 0.000,B 0.000,C 90.000,E1 273.498} C_DIS
LIN {X -0.131,Y -486.408,Z 317.517,A 0.000,B 0.000,C 90.000,E1 273.037} C_DIS
LIN {X 0.035,Y -486.494,Z 317.514,A 0.000,B 0.000,C 90.000,E1 272.522} C_DIS
LIN {X 0.207,Y -486.339,Z 317.511,A 0.000,B 0.000,C 90.000,E1 272.007} C_DIS
LIN {X 0.080,Y -485.455,Z 317.506,A 0.000,B 0.000,C 90.000,E1 271.031} C_DIS
LIN {X -0.235,Y -484.784,Z 317.503,A 0.000,B 0.000,C 90.000,E1 270.573} C_DIS
LIN {X -0.066,Y -483.838,Z 317.500,A 0.000,B 0.000,C 90.000,E1 270.057} C_DIS
LIN {X 0.097,Y -482.429,Z 317.498,A 0.000,B 0.000,C 90.000,E1 269.542} C_DIS
LIN {X -0.226,Y -480.474,Z 317.495,A 0.000,B 0.000,C 90.000,E1 269.083} C_DIS
LIN {X 0.088,Y -479.314,Z 317.493,A 0.000,B 0.000,C 90.000,E1 268.797} C_DIS
LIN {X 0.225,Y -476.299,Z 317.491,A 0.000,B 0.000,C 90.000,E1 268.282} C_DIS
LIN {X -0.115,Y -472.409,Z 317.488,A 0.000,B 0.000,C 90.000,E1 267.822} C_DIS
LIN {X 0.176,Y -470.048,Z 317.486,A 0.000,B 0.000,C 90.000,E1 267.535} C_DIS
LIN {X -0.017,Y -467.349,Z 317.485,A 0.000,B 0.000,C 90.000,E1 267.306} C_DIS
LIN {X -0.206,Y -464.292,Z 317.484,A 0.000,B 0.000,C 90.000,E1 267.078} C_DIS
LIN {X -0.103,Y -461.288,Z 317.482,A 0.000,B 0.000,C 90.000,E1 266.846} C_DIS
LIN {X -0.026,Y -457.776,Z 317.481,A 0.000,B 0.000,C 90.000,E1 266.617} C_DIS
LIN {X -0.082,Y -454.362,Z 317.480,A 0.000,B 0.000,C 90.000,E1 266.445} C_DIS
LIN {X 0.159,Y -446.795,Z 317.478,A 0.000,B 0.000,C 90.000,E1 266.102} C_DIS
LIN {X 0.139,Y -438.946,Z 317.477,A 0.000,B 0.000,C 90.000,E1 265.869} C_DIS
LIN {X 0.170,Y -429.955,Z 317.476,A 0.000,B 0.000,C 90.000,E1 265.698} C_DIS
LIN {X -0.045,Y -420.701,Z 317.476,A 0.000,B 0.000,C 90.000,E1 265.641} C_DIS
LIN {X -0.117,Y -418.326,Z 317.476,A 0.000,B 0.000,C 90.000,E1 265.641} C_DIS
LIN {X -0.083,Y -180.909,Z 317.476,A 0.000,B 0.000,C 90.000,E1 265.641} C_DIS
LIN {X 0.029,Y -180.780,Z 317.471,A 0.000,B 0.000,C 90.000,E1 264.723} C_DIS
LIN {X -0.076,Y -178.877,Z 317.443,A 0.000,B 0.000,C 90.000,E1 259.690} C_DIS
LIN {X 0.000,Y -175.919,Z 317.414,A 0.000,B 0.000,C 90.000,E1 254.574} C_DIS
LIN {X 0.056,Y -174.615,Z 317.405,A 0.000,B 0.000,C 90.000,E1 252.851} C_DIS
LIN {X -0.017,Y -171.595,Z 317.381,A 0.000,B 0.000,C 90.000,E1 248.592} C_DIS
LIN {X -0.028,Y -167.818,Z 317.357,A 0.000,B 0.000,C 90.000,E1 244.280} C_DIS
LIN {X -0.012,Y -166.541,Z 317.347,A 0.000,B 0.000,C 90.000,E1 242.538} C_DIS
LIN {X -0.100,Y -162.538,Z 317.323,A 0.000,B 0.000,C 90.000,E1 238.201} C_DIS
LIN {X -0.040,Y -161.215,Z 317.313,A 0.000,B 0.000,C 90.000,E1 236.421} C_DIS
LIN {X -0.004,Y -157.223,Z 317.289,A 0.000,B 0.000,C 90.000,E1 231.984} C_DIS
LIN {X 0.019,Y -155.948,Z 317.279,A 0.000,B 0.000,C 90.000,E1 230.194} C_DIS
LIN {X -0.022,Y -152.201,Z 317.254,A 0.000,B 0.000,C 90.000,E1 225.729} C_DIS
LIN {X -0.002,Y -150.447,Z 317.239,A 0.000,B 0.000,C 90.000,E1 223.014} C_DIS
LIN {X 0.026,Y -147.173,Z 317.214,A 0.000,B 0.000,C 90.000,E1 218.463} C_DIS
LIN {X -0.007,Y -145.190,Z 317.193,A 0.000,B 0.000,C 90.000,E1 214.818} C_DIS
LIN {X 0.027,Y -142.332,Z 317.163,A 0.000,B 0.000,C 90.000,E1 209.283} C_DIS
LIN {X -0.043,Y -141.721,Z 317.152,A 0.000,B 0.000,C 90.000,E1 207.462} C_DIS
LIN {X 0.070,Y -139.477,Z 317.116,A 0.000,B 0.000,C 90.000,E1 200.918} C_DIS
LIN {X -0.072,Y -138.974,Z 317.101,A 0.000,B 0.000,C 90.000,E1 198.181} C_DIS
LIN {X 0.050,Y -138.331,Z 317.054,A 0.000,B 0.000,C 90.000,E1 189.726} C_DIS
LIN {X 0.052,Y -139.433,Z 317.007,A 0.000,B 0.000,C 90.000,E1 181.318} C_DIS
LIN {X -0.007,Y -140.961,Z 316.976,A 0.000,B 0.000,C 90.000,E1 175.755} C_DIS
LIN {X -0.057,Y -142.717,Z 316.956,A 0.000,B 0.000,C 90.000,E1 172.064} C_DIS
LIN {X 0.042,Y -145.096,Z 316.930,A 0.000,B 0.000,C 90.000,E1 167.409} C_DIS
LIN {X 0.037,Y -147.720,Z 316.910,A 0.000,B 0.000,C 90.000,E1 163.740} C_DIS
LIN {X -0.022,Y -150.380,Z 316.889,A 0.000,B 0.000,C 90.000,E1 160.115} C_DIS
LIN {X -0.004,Y -153.809,Z 316.869,A 0.000,B 0.000,C 90.000,E1 156.485} C_DIS
LIN {X 0.055,Y -157.221,Z 316.849,A 0.000,B 0.000,C 90.000,E1 152.871} C_DIS
LIN {X -0.004,Y -161.387,Z 316.830,A 0.000,B 0.000,C 90.000,E1 149.331} C_DIS
LIN {X 0.007,Y -165.589,Z 316.810,A 0.000,B 0.000,C 90.000,E1 145.801} C_DIS
LIN {X -0.007,Y -170.512,Z 316.791,A 0.000,B 0.000,C 90.000,E1 142.316} C_DIS
LIN {X 0.037,Y -175.391,Z 316.771,A 0.000,B 0.000,C 90.000,E1 138.852} C_DIS
LIN {X -0.100,Y -181.016,Z 316.753,A 0.000,B 0.000,C 90.000,E1 135.486} C_DIS
LIN {X 0.023,Y -186.445,Z 316.734,A 0.000,B 0.000,C 90.000,E1 132.081} C_DIS
LIN {X 0.092,Y -191.070,Z 316.720,A 0.000,B 0.000,C 90.000,E1 129.564} C_DIS
LIN {X 0.015,Y -196.858,Z 316.702,A 0.000,B 0.000,C 90.000,E1 126.297} C_DIS
LIN {X -0.068,Y -200.116,Z 316.693,A 0.000,B 0.000,C 90.000,E1 124.692} C_DIS
LIN {X 0.051,Y -201.838,Z 316.687,A 0.000,B 0.000,C 90.000,E1 123.706} C_DIS
LIN {X 0.042,Y -303.335,Z 316.687,A 0.000,B 0.000,C 90.000,E1 123.706} C_DIS
LIN {X 0.020,Y -305.740,Z 316.687,A 0.000,B 0.000,C 90.000,E1 123.658} C_DIS
LIN {X -0.076,Y -310.898,Z 316.685,A 0.000,B 0.000,C 90.000,E1 123.372} C_DIS
LIN {X 0.089,Y -313.768,Z 316.684,A 0.000,B 0.000,C 90.000,E1 123.038} C_DIS
LIN {X 0.049,Y -315.797,Z 316.682,A 0.000,B 0.000,C 90.000,E1 122.752} C_DIS
LIN {X 0.007,Y -317.388,Z 316.680,A 0.000,B 0.000,C 90.000,E1 122.467} C_DIS
LIN {X 0.143,Y -319.927,Z 316.677,A 0.000,B 0.000,C 90.000,E1 121.799} C_DIS
LIN {X 0.095,Y -330.905,Z 316.661,A 0.000,B 0.000,C 90.000,E1 118.949} C_DIS
LIN {X 0.031,Y -343.294,Z 316.645,A 0.000,B 0.000,C 90.000,E1 116.155} C_DIS
LIN {X 0.141,Y -355.577,Z 316.632,A 0.000,B 0.000,C 90.000,E1 113.695} C_DIS
LIN {X -0.054,Y -369.150,Z 316.618,A 0.000,B 0.000,C 90.000,E1 111.334} C_DIS
LIN {X 0.170,Y -384.113,Z 316.605,A 0.000,B 0.000,C 90.000,E1 108.960} C_DIS
LIN {X 0.172,Y -400.575,Z 316.593,A 0.000,B 0.000,C 90.000,E1 106.677} C_DIS
LIN {X -0.032,Y -418.661,Z 316.580,A 0.000,B 0.000,C 90.000,E1 104.481} C_DIS
LIN {X -0.193,Y -438.335,Z 316.569,A 0.000,B 0.000,C 90.000,E1 102.355} C_DIS
LIN {X -0.130,Y -458.730,Z 316.557,A 0.000,B 0.000,C 90.000,E1 100.366} C_DIS
LIN {X -0.176,Y -482.276,Z 316.546,A 0.000,B 0.000,C 90.000,E1 98.341} C_DIS
LIN {X -0.205,Y -495.619,Z 316.540,A 0.000,B 0.000,C 90.000,E1 97.296} C_DIS
LIN {X 0.251,Y -499.535,Z 316.538,A 0.000,B 0.000,C 90.000,E1 96.834} C_DIS
LIN {X 0.104,Y -501.090,Z 316.537,A 0.000,B 0.000,C 90.000,E1 96.606} C_DIS
LIN {X 0.014,Y -502.251,Z 316.535,A 0.000,B 0.000,C 90.000,E1 96.372} C_DIS
LIN {X -0.194,Y -503.628,Z 316.533,A 0.000,B 0.000,C 90.000,E1 95.910} C_DIS
LIN {X 0.103,Y -503.951,Z 316.530,A 0.000,B 0.000,C 90.000,E1 95.391} C_DIS
LIN {X -0.138,Y -503.274,Z 316.527,A 0.000,B 0.000,C 90.000,E1 94.935} C_DIS
LIN {X 0.170,Y -501.475,Z 316.525,A 0.000,B 0.000,C 90.000,E1 94.416} C_DIS
LIN {X 0.052,Y -500.045,Z 316.523,A 0.000,B 0.000,C 90.000,E1 94.188} C_DIS
LIN {X 0.215,Y -494.558,Z 316.519,A 0.000,B 0.000,C 90.000,E1 93.440} C_DIS
LIN {X 0.180,Y -486.641,Z 316.514,A 0.000,B 0.000,C 90.000,E1 92.465} C_DIS
LIN {X -0.171,Y -470.156,Z 316.503,A 0.000,B 0.000,C 90.000,E1 90.516} C_DIS
LIN {X -0.188,Y -452.748,Z 316.490,A 0.000,B 0.000,C 90.000,E1 88.224} C_DIS
LIN {X 0.183,Y -433.486,Z 316.474,A 0.000,B 0.000,C 90.000,E1 85.298} C_DIS
LIN {X -0.076,Y -417.719,Z 316.459,A 0.000,B 0.000,C 90.000,E1 82.648} C_DIS
LIN {X 0.220,Y -403.209,Z 316.444,A 0.000,B 0.000,C 90.000,E1 79.859} C_DIS
LIN {X -0.111,Y -394.559,Z 316.435,A 0.000,B 0.000,C 90.000,E1 78.229} C_DIS
LIN {X 0.000,Y -384.398,Z 316.423,A 0.000,B 0.000,C 90.000,E1 76.228} C_DIS
LIN {X -0.002,Y -372.865,Z 316.411,A 0.000,B 0.000,C 90.000,E1 73.921} C_DIS
LIN {X -0.041,Y -362.715,Z 316.399,A 0.000,B 0.000,C 90.000,E1 71.873} C_DIS
LIN {X 0.159,Y -352.536,Z 316.388,A 0.000,B 0.000,C 90.000,E1 69.752} C_DIS
LIN {X -0.039,Y -338.373,Z 316.371,A 0.000,B 0.000,C 90.000,E1 66.741} C_DIS
LIN {X -0.184,Y -328.289,Z 316.357,A 0.000,B 0.000,C 90.000,E1 64.280} C_DIS
LIN {X 0.006,Y -318.889,Z 316.343,A 0.000,B 0.000,C 90.000,E1 61.719} C_DIS
LIN {X 0.032,Y -308.817,Z 316.327,A 0.000,B 0.000,C 90.000,E1 58.820} C_DIS
LIN {X 0.034,Y -298.164,Z 316.309,A 0.000,B 0.000,C 90.000,E1 55.548} C_DIS
LIN {X 0.161,Y -288.227,Z 316.290,A 0.000,B 0.000,C 90.000,E1 52.190} C_DIS
LIN {X -0.140,Y -280.492,Z 316.275,A 0.000,B 0.000,C 90.000,E1 49.542} C_DIS
LIN {X -0.086,Y -272.675,Z 316.260,A 0.000,B 0.000,C 90.000,E1 46.782} C_DIS
LIN {X 0.131,Y -265.085,Z 316.244,A 0.000,B 0.000,C 90.000,E1 43.947} C_DIS
LIN {X 0.082,Y -259.498,Z 316.233,A 0.000,B 0.000,C 90.000,E1 41.838} C_DIS
LIN {X 0.018,Y -251.921,Z 316.217,A 0.000,B 0.000,C 90.000,E1 38.991} C_DIS
LIN {X 0.136,Y -246.192,Z 316.205,A 0.000,B 0.000,C 90.000,E1 36.790} C_DIS
LIN {X 0.044,Y -240.226,Z 316.192,A 0.000,B 0.000,C 90.000,E1 34.612} C_DIS
LIN {X -0.104,Y -230.543,Z 316.172,A 0.000,B 0.000,C 90.000,E1 30.924} C_DIS
LIN {X 0.077,Y -223.123,Z 316.155,A 0.000,B 0.000,C 90.000,E1 27.847} C_DIS
LIN {X 0.061,Y -216.455,Z 316.138,A 0.000,B 0.000,C 90.000,E1 24.771} C_DIS
LIN {X 0.008,Y -210.644,Z 316.120,A 0.000,B 0.000,C 90.000,E1 21.663} C_DIS
LIN {X 0.056,Y -205.583,Z 316.103,A 0.000,B 0.000,C 90.000,E1 18.489} C_DIS
LIN {X 0.035,Y -201.320,Z 316.085,A 0.000,B 0.000,C 90.000,E1 15.300} C_DIS
LIN {X -0.077,Y -196.921,Z 316.063,A 0.000,B 0.000,C 90.000,E1 11.299} C_DIS
LIN {X 0.077,Y -193.579,Z 316.040,A 0.000,B 0.000,C 90.000,E1 7.182} C_DIS
LIN {X 0.089,Y -190.634,Z 316.008,A 0.000,B 0.000,C 90.000,E1 1.432} C_DIS
LIN {X -0.089,Y -191.792,Z 315.929,A 0.000,B 0.000,C 90.000,E1 347.173} C_DIS
LIN {X -0.051,Y -195.135,Z 315.901,A 0.000,B 0.000,C 90.000,E1 342.236} C_DIS
LIN {X -0.035,Y -199.060,Z 315.879,A 0.000,B 0.000,C 90.000,E1 338.156} C_DIS
LIN {X 0.027,Y -203.982,Z 315.856,A 0.000,B 0.000,C 90.000,E1 334.101} C_DIS
LIN {X -0.040,Y -209.996,Z 315.834,A 0.000,B 0.000,C 90.000,E1 330.127} C_DIS
LIN {X 0.038,Y -216.781,Z 315.812,A 0.000,B 0.000,C 90.000,E1 326.167} C_DIS
LIN {X 0.066,Y -222.827,Z 315.795,A 0.000,B 0.000,C 90.000,E1 323.050} C_DIS
LIN {X 0.031,Y -229.639,Z 315.778,A 0.000,B 0.000,C 90.000,E1 319.989} C_DIS
LIN {X -0.058,Y -237.496,Z 315.761,A 0.000,B 0.000,C 90.000,E1 316.986} C_DIS
LIN {X -0.110,Y -246.466,Z 315.744,A 0.000,B 0.000,C 90.000,E1 314.028} C_DIS
LIN {X 0.113,Y -257.691,Z 315.726,A 0.000,B 0.000,C 90.000,E1 310.701} C_DIS
LIN {X -0.005,Y -269.836,Z 315.708,A 0.000,B 0.000,C 90.000,E1 307.523} C_DIS
LIN {X -0.051,Y -283.269,Z 315.691,A 0.000,B 0.000,C 90.000,E1 304.405} C_DIS
LIN {X 0.059,Y -294.793,Z 315.678,A 0.000,B 0.000,C 90.000,E1 302.005} C_DIS
LIN {X 0.047,Y -311.229,Z 315.661,A 0.000,B 0.000,C 90.000,E1 299.027} C_DIS
LIN {X -0.108,Y -325.346,Z 315.649,A 0.000,B 0.000,C 90.000,E1 296.796} C_DIS
LIN {X 0.028,Y -342.664,Z 315.635,A 0.000,B 0.000,C 90.000,E1 294.259} C_DIS
LIN {X -0.126,Y -360.561,Z 315.621,A 0.000,B 0.000,C 90.000,E1 291.844} C_DIS
LIN {X 0.037,Y -378.807,Z 315.608,A 0.000,B 0.000,C 90.000,E1 289.450} C_DIS
LIN {X 0.042,Y -398.001,Z 315.595,A 0.000,B 0.000,C 90.000,E1 287.149} C_DIS
LIN {X -0.049,Y -412.443,Z 315.586,A 0.000,B 0.000,C 90.000,E1 285.481} C_DIS
LIN {X -0.130,Y -424.395,Z 315.578,A 0.000,B 0.000,C 90.000,E1 284.120} C_DIS
LIN {X 0.104,Y -433.436,Z 315.572,A 0.000,B 0.000,C 90.000,E1 283.008} C_DIS
LIN {X 0.030,Y -441.593,Z 315.566,A 0.000,B 0.000,C 90.000,E1 281.951} C_DIS
LIN {X 0.049,Y -449.141,Z 315.561,A 0.000,B 0.000,C 90.000,E1 280.894} C_DIS
LIN {X 0.072,Y -456.025,Z 315.555,A 0.000,B 0.000,C 90.000,E1 279.849} C_DIS
LIN {X 0.179,Y -462.400,Z 315.549,A 0.000,B 0.000,C 90.000,E1 278.803} C_DIS
LIN {X 0.135,Y -469.785,Z 315.542,A 0.000,B 0.000,C 90.000,E1 277.530} C_DIS
LIN {X -0.073,Y -475.361,Z 315.536,A 0.000,B 0.000,C 90.000,E1 276.543} C_DIS
LIN {X -0.141,Y -479.102,Z 315.532,A 0.000,B 0.000,C 90.000,E1 275.796} C_DIS
LIN {X 0.147,Y -480.263,Z 315.531,A 0.000,B 0.000,C 90.000,E1 275.511} C_DIS
LIN {X -0.175,Y -482.249,Z 315.528,A 0.000,B 0.000,C 90.000,E1 275.049} C_DIS
LIN {X -0.012,Y -483.855,Z 315.525,A 0.000,B 0.000,C 90.000,E1 274.531} C_DIS
LIN {X 0.161,Y -485.075,Z 315.522,A 0.000,B 0.000,C 90.000,E1 274.012} C_DIS
LIN {X -0.173,Y -485.901,Z 315.520,A 0.000,B 0.000,C 90.000,E1 273.555} C_DIS
LIN {X 0.013,Y -486.338,Z 315.517,A 0.000,B 0.000,C 90.000,E1 273.037} C_DIS
LIN {X 0.178,Y -486.441,Z 315.514,A 0.000,B 0.000,C 90.000,E1 272.522} C_DIS
LIN {X -0.136,Y -486.281,Z 315.511,A 0.000,B 0.000,C 90.000,E1 272.064} C_DIS
LIN {X 0.051,Y -485.946,Z 315.509,A 0.000,B 0.000,C 90.000,E1 271.547} C_DIS
LIN {X -0.093,Y -484.736,Z 315.503,A 0.000,B 0.000,C 90.000,E1 270.573} C_DIS
LIN {X 0.075,Y -483.821,Z 315.500,A 0.000,B 0.000,C 90.000,E1 270.057} C_DIS
LIN {X 0.238,Y -482.427,Z 315.498,A 0.000,B 0.000,C 90.000,E1 269.542} C_DIS
LIN {X -0.086,Y -480.533,Z 315.495,A 0.000,B 0.000,C 90.000,E1 269.083} C_DIS
LIN {X 0.061,Y -478.023,Z 315.492,A 0.000,B 0.000,C 90.000,E1 268.568} C_DIS
LIN {X 0.204,Y -474.646,Z 315.489,A 0.000,B 0.000,C 90.000,E1 268.051} C_DIS
LIN {X -0.157,Y -470.299,Z 315.487,A 0.000,B 0.000,C 90.000,E1 267.593} C_DIS
LIN {X 0.121,Y -467.676,Z 315.485,A 0.000,B 0.000,C 90.000,E1 267.306} C_DIS
LIN {X 0.034,Y -461.685,Z 315.483,A 0.000,B 0.000,C 90.000,E1 266.846} C_DIS
LIN {X 0.113,Y -458.253,Z 315.481,A 0.000,B 0.000,C 90.000,E1 266.617} C_DIS
LIN {X -0.049,Y -450.839,Z 315.479,A 0.000,B 0.000,C 90.000,E1 266.274} C_DIS
LIN {X 0.019,Y -443.224,Z 315.478,A 0.000,B 0.000,C 90.000,E1 265.988} C_DIS
LIN {X 0.207,Y -434.648,Z 315.477,A 0.000,B 0.000,C 90.000,E1 265.755} C_DIS
LIN {X 0.121,Y -430.544,Z 315.476,A 0.000,B 0.000,C 90.000,E1 265.698} C_DIS
LIN {X -0.114,Y -421.405,Z 315.476,A 0.000,B 0.000,C 90.000,E1 265.641} C_DIS
LIN {X 0.155,Y -416.859,Z 315.476,A 0.000,B 0.000,C 90.000,E1 265.584} C_DIS
LIN {X 0.035,Y -180.908,Z 315.476,A 0.000,B 0.000,C 90.000,E1 265.584} C_DIS
LIN {X -0.004,Y -180.776,Z 315.471,A 0.000,B 0.000,C 90.000,E1 264.723} C_DIS
LIN {X 0.067,Y -178.872,Z 315.443,A 0.000,B 0.000,C 90.000,E1 259.634} C_DIS
LIN {X -0.032,Y -175.915,Z 315.414,A 0.000,B 0.000,C 90.000,E1 254.574} C_DIS
LIN {X 0.024,Y -174.606,Z 315.405,A 0.000,B 0.000,C 90.000,E1 252.851} C_DIS
LIN {X -0.050,Y -171.588,Z 315.381,A 0.000,B 0.000,C 90.000,E1 248.592} C_DIS
LIN {X -0.060,Y -167.810,Z 315.357,A 0.000,B 0.000,C 90.000,E1 244.280} C_DIS
LIN {X -0.043,Y -166.531,Z 315.347,A 0.000,B 0.000,C 90.000,E1 242.538} C_DIS
LIN {X 0.092,Y -162.530,Z 315.323,A 0.000,B 0.000,C 90.000,E1 238.122} C_DIS
LIN {X -0.071,Y -161.205,Z 315.313,A 0.000,B 0.000,C 90.000,E1 236.421} C_DIS
LIN {X -0.035,Y -157.214,Z 315.289,A 0.000,B 0.000,C 90.000,E1 231.984} C_DIS
LIN {X -0.012,Y -155.940,Z 315.279,A 0.000,B 0.000,C 90.000,E1 230.194} C_DIS
LIN {X -0.053,Y -152.193,Z 315.254,A 0.000,B 0.000,C 90.000,E1 225.729} C_DIS
LIN {X -0.031,Y -150.439,Z 315.239,A 0.000,B 0.000,C 90.000,E1 223.014} C_DIS
LIN {X -0.003,Y -147.166,Z 315.214,A 0.000,B 0.000,C 90.000,E1 218.463} C_DIS
LIN {X -0.037,Y -145.181,Z 315.193,A 0.000,B 0.000,C 90.000,E1 214.818} C_DIS
LIN {X -0.002,Y -142.327,Z 315.163,A 0.000,B 0.000,C 90.000,E1 209.283} C_DIS
LIN {X -0.006,Y -141.716,Z 315.152,A 0.000,B 0.000,C 90.000,E1 207.436} C_DIS
LIN {X 0.042,Y -139.474,Z 315.116,A 0.000,B 0.000,C 90.000,E1 200.918} C_DIS
LIN {X 0.032,Y -138.971,Z 315.101,A 0.000,B 0.000,C 90.000,E1 198.127} C_DIS
LIN {X 0.021,Y -138.330,Z 315.054,A 0.000,B 0.000,C 90.000,E1 189.726} C_DIS
LIN {X 0.024,Y -139.436,Z 315.007,A 0.000,B 0.000,C 90.000,E1 181.318} C_DIS
LIN {X -0.036,Y -140.965,Z 314.976,A 0.000,B 0.000,C 90.000,E1 175.755} C_DIS
LIN {X 0.055,Y -142.722,Z 314.956,A 0.000,B 0.000,C 90.000,E1 172.008} C_DIS
LIN {X 0.013,Y -145.104,Z 314.930,A 0.000,B 0.000,C 90.000,E1 167.409} C_DIS
LIN {X 0.008,Y -147.728,Z 314.910,A 0.000,B 0.000,C 90.000,E1 163.740} C_DIS
LIN {X -0.052,Y -150.388,Z 314.889,A 0.000,B 0.000,C 90.000,E1 160.115} C_DIS
LIN {X -0.034,Y -153.821,Z 314.869,A 0.000,B 0.000,C 90.000,E1 156.485} C_DIS
LIN {X 0.025,Y -157.233,Z 314.849,A 0.000,B 0.000,C 90.000,E1 152.871} C_DIS
LIN {X -0.035,Y -161.401,Z 314.830,A 0.000,B 0.000,C 90.000,E1 149.331} C_DIS
LIN {X -0.024,Y -165.604,Z 314.810,A 0.000,B 0.000,C 90.000,E1 145.801} C_DIS
LIN {X -0.039,Y -170.529,Z 314.791,A 0.000,B 0.000,C 90.000,E1 142.316} C_DIS
LIN {X 0.005,Y -175.408,Z 314.771,A 0.000,B 0.000,C 90.000,E1 138.852} C_DIS
LIN {X -0.004,Y -181.032,Z 314.752,A 0.000,B 0.000,C 90.000,E1 135.445} C_DIS
LIN {X -0.011,Y -186.465,Z 314.734,A 0.000,B 0.000,C 90.000,E1 132.081} C_DIS
LIN {X 0.058,Y -191.087,Z 314.720,A 0.000,B 0.000,C 90.000,E1 129.564} C_DIS
LIN {X -0.021,Y -196.878,Z 314.702,A 0.000,B 0.000,C 90.000,E1 126.297} C_DIS
LIN {X 0.011,Y -200.137,Z 314.693,A 0.000,B 0.000,C 90.000,E1 124.659} C_DIS
LIN {X -0.089,Y -201.907,Z 314.687,A 0.000,B 0.000,C 90.000,E1 123.706} C_DIS
LIN {X 0.067,Y -303.229,Z 314.687,A 0.000,B 0.000,C 90.000,E1 123.658} C_DIS
LIN {X -0.035,Y -304.578,Z 314.687,A 0.000,B 0.000,C 90.000,E1 123.658} C_DIS
LIN {X 0.003,Y -308.458,Z 314.686,A 0.000,B 0.000,C 90.000,E1 123.499} C_DIS
LIN {X -0.131,Y -310.628,Z 314.685,A 0.000,B 0.000,C 90.000,E1 123.372} C_DIS
LIN {X 0.033,Y -313.630,Z 314.684,A 0.000,B 0.000,C 90.000,E1 123.038} C_DIS
LIN {X 0.059,Y -317.259,Z 314.680,A 0.000,B 0.000,C 90.000,E1 122.467} C_DIS
LIN {X 0.121,Y -318.703,Z 314.679,A 0.000,B 0.000,C 90.000,E1 122.133} C_DIS
LIN {X 0.134,Y -330.856,Z 314.661,A 0.000,B 0.000,C 90.000,E1 118.949} C_DIS
LIN {X 0.071,Y -343.240,Z 314.645,A 0.000,B 0.000,C 90.000,E1 116.155} C_DIS
LIN {X 0.038,Y -355.520,Z 314.632,A 0.000,B 0.000,C 90.000,E1 113.718} C_DIS
LIN {X -0.150,Y -369.089,Z 314.618,A 0.000,B 0.000,C 90.000,E1 111.354} C_DIS
LIN {X 0.210,Y -384.048,Z 314.605,A 0.000,B 0.000,C 90.000,E1 108.960} C_DIS
LIN {X 0.211,Y -400.506,Z 314.593,A 0.000,B 0.000,C 90.000,E1 106.677} C_DIS
LIN {X 0.008,Y -418.587,Z 314.580,A 0.000,B 0.000,C 90.000,E1 104.481} C_DIS
LIN {X -0.154,Y -438.257,Z 314.569,A 0.000,B 0.000,C 90.000,E1 102.355} C_DIS
LIN {X -0.095,Y -458.651,Z 314.558,A 0.000,B 0.000,C 90.000,E1 100.366} C_DIS
LIN {X -0.143,Y -482.196,Z 314.546,A 0.000,B 0.000,C 90.000,E1 98.341} C_DIS
LIN {X -0.174,Y -495.547,Z 314.540,A 0.000,B 0.000,C 90.000,E1 97.296} C_DIS
LIN {X -0.207,Y -499.585,Z 314.538,A 0.000,B 0.000,C 90.000,E1 96.891} C_DIS
LIN {X 0.154,Y -501.177,Z 314.537,A 0.000,B 0.000,C 90.000,E1 96.606} C_DIS
LIN {X 0.075,Y -502.371,Z 314.535,A 0.000,B 0.000,C 90.000,E1 96.372} C_DIS
LIN {X -0.132,Y -503.811,Z 314.533,A 0.000,B 0.000,C 90.000,E1 95.910} C_DIS
LIN {X 0.166,Y -504.187,Z 314.530,A 0.000,B 0.000,C 90.000,E1 95.391} C_DIS
LIN {X -0.073,Y -503.561,Z 314.527,A 0.000,B 0.000,C 90.000,E1 94.935} C_DIS
LIN {X 0.235,Y -501.826,Z 314.525,A 0.000,B 0.000,C 90.000,E1 94.416} C_DIS
LIN {X 0.117,Y -500.439,Z 314.523,A 0.000,B 0.000,C 90.000,E1 94.188} C_DIS
LIN {X -0.211,Y -495.009,Z 314.519,A 0.000,B 0.000,C 90.000,E1 93.498} C_DIS
LIN {X -0.234,Y -487.074,Z 314.514,A 0.000,B 0.000,C 90.000,E1 92.522} C_DIS
LIN {X 0.086,Y -472.589,Z 314.504,A 0.000,B 0.000,C 90.000,E1 90.745} C_DIS
LIN {X -0.102,Y -453.101,Z 314.490,A 0.000,B 0.000,C 90.000,E1 88.224} C_DIS
LIN {X -0.156,Y -433.799,Z 314.474,A 0.000,B 0.000,C 90.000,E1 85.355} C_DIS
LIN {X 0.022,Y -418.024,Z 314.459,A 0.000,B 0.000,C 90.000,E1 82.648} C_DIS
LIN {X -0.048,Y -402.079,Z 314.442,A 0.000,B 0.000,C 90.000,E1 79.634} C_DIS
LIN {X 0.066,Y -393.412,Z 314.433,A 0.000,B 0.000,C 90.000,E1 77.937} C_DIS
LIN {X 0.151,Y -383.249,Z 314.422,A 0.000,B 0.000,C 90.000,E1 75.936} C_DIS
LIN {X 0.111,Y -373.173,Z 314.411,A 0.000,B 0.000,C 90.000,E1 73.921} C_DIS
LIN {X 0.077,Y -363.028,Z 314.399,A 0.000,B 0.000,C 90.000,E1 71.873} C_DIS
LIN {X -0.050,Y -352.864,Z 314.388,A 0.000,B 0.000,C 90.000,E1 69.806} C_DIS
LIN {X 0.089,Y -337.397,Z 314.369,A 0.000,B 0.000,C 90.000,E1 66.433} C_DIS
LIN {X 0.019,Y -326.248,Z 314.354,A 0.000,B 0.000,C 90.000,E1 63.640} C_DIS
LIN {X -0.128,Y -316.956,Z 314.339,A 0.000,B 0.000,C 90.000,E1 61.129} C_DIS
LIN {X -0.042,Y -308.069,Z 314.325,A 0.000,B 0.000,C 90.000,E1 58.535} C_DIS
LIN {X 0.134,Y -296.465,Z 314.305,A 0.000,B 0.000,C 90.000,E1 54.895} C_DIS
LIN {X -0.014,Y -286.610,Z 314.287,A 0.000,B 0.000,C 90.000,E1 51.582} C_DIS
LIN {X 0.015,Y -280.785,Z 314.275,A 0.000,B 0.000,C 90.000,E1 49.542} C_DIS
LIN {X 0.073,Y -272.940,Z 314.260,A 0.000,B 0.000,C 90.000,E1 46.782} C_DIS
LIN {X -0.083,Y -265.346,Z 314.245,A 0.000,B 0.000,C 90.000,E1 44.028} C_DIS
LIN {X -0.123,Y -259.769,Z 314.233,A 0.000,B 0.000,C 90.000,E1 41.919} C_DIS
LIN {X -0.014,Y -252.194,Z 314.217,A 0.000,B 0.000,C 90.000,E1 39.036} C_DIS
LIN {X -0.045,Y -246.483,Z 314.205,A 0.000,B 0.000,C 90.000,E1 36.870} C_DIS
LIN {X 0.014,Y -240.528,Z 314.193,A 0.000,B 0.000,C 90.000,E1 34.659} C_DIS
LIN {X 0.065,Y -230.823,Z 314.172,A 0.000,B 0.000,C 90.000,E1 30.924} C_DIS
LIN {X 0.049,Y -223.386,Z 314.155,A 0.000,B 0.000,C 90.000,E1 27.897} C_DIS
LIN {X 0.036,Y -216.730,Z 314.138,A 0.000,B 0.000,C 90.000,E1 24.823} C_DIS
LIN {X -0.014,Y -210.907,Z 314.121,A 0.000,B 0.000,C 90.000,E1 21.716} C_DIS
LIN {X 0.036,Y -205.820,Z 314.103,A 0.000,B 0.000,C 90.000,E1 18.544} C_DIS
LIN {X 0.076,Y -200.615,Z 314.081,A 0.000,B 0.000,C 90.000,E1 14.537} C_DIS
LIN {X -0.094,Y -196.414,Z 314.058,A 0.000,B 0.000,C 90.000,E1 10.546} C_DIS
LIN {X 0.046,Y -193.272,Z 314.036,A 0.000,B 0.000,C 90.000,E1 6.429} C_DIS
LIN {X 0.019,Y -190.560,Z 314.004,A 0.000,B 0.000,C 90.000,E1 0.688} C_DIS
LIN {X -0.075,Y -191.920,Z 313.929,A 0.000,B 0.000,C 90.000,E1 347.173} C_DIS
LIN {X -0.033,Y -195.256,Z 313.901,A 0.000,B 0.000,C 90.000,E1 342.236} C_DIS
LIN {X -0.012,Y -199.158,Z 313.879,A 0.000,B 0.000,C 90.000,E1 338.156} C_DIS
LIN {X 0.054,Y -204.069,Z 313.856,A 0.000,B 0.000,C 90.000,E1 334.101} C_DIS
LIN {X -0.010,Y -210.065,Z 313.834,A 0.000,B 0.000,C 90.000,E1 330.127} C_DIS
LIN {X 0.071,Y -216.825,Z 313.812,A 0.000,B 0.000,C 90.000,E1 326.167} C_DIS
LIN {X 0.101,Y -222.871,Z 313.795,A 0.000,B 0.000,C 90.000,E1 323.050} C_DIS
LIN {X 0.068,Y -229.699,Z 313.778,A 0.000,B 0.000,C 90.000,E1 319.989} C_DIS
LIN {X -0.017,Y -237.599,Z 313.761,A 0.000,B 0.000,C 90.000,E1 316.986} C_DIS
LIN {X -0.066,Y -246.598,Z 313.745,A 0.000,B 0.000,C 90.000,E1 314.028} C_DIS
LIN {X -0.031,Y -257.826,Z 313.726,A 0.000,B 0.000,C 90.000,E1 310.744} C_DIS
LIN {X 0.051,Y -269.997,Z 313.709,A 0.000,B 0.000,C 90.000,E1 307.523} C_DIS
LIN {X 0.014,Y -283.439,Z 313.691,A 0.000,B 0.000,C 90.000,E1 304.405} C_DIS
LIN {X 0.131,Y -294.991,Z 313.678,A 0.000,B 0.000,C 90.000,E1 302.005} C_DIS
LIN {X -0.144,Y -311.463,Z 313.661,A 0.000,B 0.000,C 90.000,E1 299.077} C_DIS
LIN {X -0.017,Y -325.616,Z 313.649,A 0.000,B 0.000,C 90.000,E1 296.796} C_DIS
LIN {X 0.131,Y -342.925,Z 313.635,A 0.000,B 0.000,C 90.000,E1 294.259} C_DIS
LIN {X -0.011,Y -360.804,Z 313.621,A 0.000,B 0.000,C 90.000,E1 291.844} C_DIS
LIN {X 0.164,Y -378.990,Z 313.608,A 0.000,B 0.000,C 90.000,E1 289.450} C_DIS
LIN {X 0.017,Y -395.694,Z 313.597,A 0.000,B 0.000,C 90.000,E1 287.457} C_DIS
LIN {X -0.112,Y -410.097,Z 313.588,A 0.000,B 0.000,C 90.000,E1 285.788} C_DIS
LIN {X -0.125,Y -422.027,Z 313.580,A 0.000,B 0.000,C 90.000,E1 284.411} C_DIS
LIN {X -0.087,Y -428.966,Z 313.575,A 0.000,B 0.000,C 90.000,E1 283.592} C_DIS
LIN {X 0.013,Y -435.455,Z 313.571,A 0.000,B 0.000,C 90.000,E1 282.771} C_DIS
LIN {X -0.039,Y -443.408,Z 313.565,A 0.000,B 0.000,C 90.000,E1 281.715} C_DIS
LIN {X -0.002,Y -450.816,Z 313.559,A 0.000,B 0.000,C 90.000,E1 280.658} C_DIS
LIN {X -0.144,Y -459.108,Z 313.552,A 0.000,B 0.000,C 90.000,E1 279.378} C_DIS
LIN {X -0.077,Y -465.232,Z 313.546,A 0.000,B 0.000,C 90.000,E1 278.341} C_DIS
LIN {X -0.082,Y -472.426,Z 313.539,A 0.000,B 0.000,C 90.000,E1 277.068} C_DIS
LIN {X 0.157,Y -477.680,Z 313.534,A 0.000,B 0.000,C 90.000,E1 276.030} C_DIS
LIN {X -0.177,Y -480.051,Z 313.531,A 0.000,B 0.000,C 90.000,E1 275.568} C_DIS
LIN {X -0.020,Y -482.068,Z 313.528,A 0.000,B 0.000,C 90.000,E1 275.049} C_DIS
LIN {X 0.142,Y -483.687,Z 313.525,A 0.000,B 0.000,C 90.000,E1 274.531} C_DIS
LIN {X -0.170,Y -484.935,Z 313.522,A 0.000,B 0.000,C 90.000,E1 274.069} C_DIS
LIN {X -0.022,Y -485.784,Z 313.520,A 0.000,B 0.000,C 90.000,E1 273.555} C_DIS
LIN {X 0.164,Y -486.280,Z 313.517,A 0.000,B 0.000,C 90.000,E1 273.037} C_DIS
LIN {X -0.157,Y -486.377,Z 313.514,A 0.000,B 0.000,C 90.000,E1 272.579} C_DIS
LIN {X 0.014,Y -486.243,Z 313.511,A 0.000,B 0.000,C 90.000,E1 272.064} C_DIS
LIN {X 0.201,Y -485.890,Z 313.509,A 0.000,B 0.000,C 90.000,E1 271.547} C_DIS
LIN {X 0.056,Y -484.683,Z 313.503,A 0.000,B 0.000,C 90.000,E1 270.573} C_DIS
LIN {X 0.223,Y -483.785,Z 313.500,A 0.000,B 0.000,C 90.000,E1 270.057} C_DIS
LIN {X -0.097,Y -482.460,Z 313.498,A 0.000,B 0.000,C 90.000,E1 269.599} C_DIS
LIN {X 0.060,Y -480.639,Z 313.495,A 0.000,B 0.000,C 90.000,E1 269.083} C_DIS
LIN {X 0.208,Y -478.141,Z 313.492,A 0.000,B 0.000,C 90.000,E1 268.568} C_DIS
LIN {X -0.125,Y -474.875,Z 313.489,A 0.000,B 0.000,C 90.000,E1 268.108} C_DIS
LIN {X 0.169,Y -472.887,Z 313.488,A 0.000,B 0.000,C 90.000,E1 267.822} C_DIS
LIN {X -0.201,Y -467.987,Z 313.485,A 0.000,B 0.000,C 90.000,E1 267.364} C_DIS
LIN {X 0.129,Y -462.048,Z 313.483,A 0.000,B 0.000,C 90.000,E1 266.849} C_DIS
LIN {X 0.207,Y -458.619,Z 313.481,A 0.000,B 0.000,C 90.000,E1 266.617} C_DIS
LIN {X 0.108,Y -455.281,Z 313.480,A 0.000,B 0.000,C 90.000,E1 266.445} C_DIS
LIN {X -0.194,Y -447.930,Z 313.479,A 0.000,B 0.000,C 90.000,E1 266.159} C_DIS
LIN {X 0.140,Y -440.143,Z 313.477,A 0.000,B 0.000,C 90.000,E1 265.869} C_DIS
LIN {X 0.081,Y -431.310,Z 313.476,A 0.000,B 0.000,C 90.000,E1 265.698} C_DIS
LIN {X -0.034,Y -424.527,Z 313.476,A 0.000,B 0.000,C 90.000,E1 265.641} C_DIS
LIN {X 0.046,Y -416.511,Z 313.475,A 0.000,B 0.000,C 90.000,E1 265.584} C_DIS
LIN {X -0.009,Y -180.908,Z 313.475,A 0.000,B 0.000,C 90.000,E1 265.584} C_DIS
LIN {X 0.010,Y -180.700,Z 313.470,A 0.000,B 0.000,C 90.000,E1 264.546} C_DIS
LIN {X 0.019,Y -179.030,Z 313.445,A 0.000,B 0.000,C 90.000,E1 260.151} C_DIS
LIN {X -0.095,Y -178.682,Z 313.441,A 0.000,B 0.000,C 90.000,E1 259.342} C_DIS
LIN {X 0.016,Y -175.732,Z 313.412,A 0.000,B 0.000,C 90.000,E1 254.212} C_DIS
LIN {X 0.012,Y -171.917,Z 313.384,A 0.000,B 0.000,C 90.000,E1 249.082} C_DIS
LIN {X -0.013,Y -171.284,Z 313.379,A 0.000,B 0.000,C 90.000,E1 248.230} C_DIS
